LIN {X 0,Y 304.273,Z 903.558,A -85,B 0,C 180,E1 11483.308,E2 11483.308} C_VEL
LIN {X 0,Y 294.742,Z 920.406,A -85,B 0,C 180,E1 11480.364,E2 11480.364} C_VEL
LIN {X 0,Y 285.565,Z 936.169,A -85,B 0,C 180,E1 11477.041,E2 11477.041} C_VEL
LIN {X 0,Y 276.52,Z 951.203,A -85,B 0,C 180,E1 11473.115,E2 11473.115} C_VEL
LIN {X 0,Y 268.033,Z 965.419,A -85,B 0,C 180,E1 11468.539,E2 11468.539} C_VEL
LIN {X 0,Y 261.444,Z 977.018,A -85,B 0,C 180,E1 11463.948,E2 11463.948} C_VEL
LIN {X 0,Y 256.111,Z 986.967,A -85,B 0,C 180,E1 11459.016,E2 11459.016} C_VEL
LIN {X 0,Y 252.21,Z 995.391,A -85,B 0,C 180,E1 11453.857,E2 11453.857} C_VEL
LIN {X 0,Y 249.926,Z 1001.381,A -85,B 0,C 180,E1 11449.156,E2 11449.156} C_VEL
LIN {X 0,Y 248.555,Z 1006.524,A -85,B 0,C 180,E1 11443.973,E2 11443.973} C_VEL
LIN {X 0,Y 248.056,Z 1009.801,A -85,B 0,C 180,E1 11439.05,E2 11439.05} C_VEL
LIN {X 0,Y 247.979,Z 1011.619,A -85,B 0,C 180,E1 11434.631,E2 11434.631} C_VEL
LIN {X 0,Y 248.01,Z 1012.279,A -85,B 0,C 180,E1 11430.006,E2 11430.006} C_VEL
LIN {X 0,Y 247.985,Z 1011.616,A -85,B 0,C 180,E1 11425.613,E2 11425.613} C_VEL
LIN {X 0,Y 248.04,Z 1010.062,A -85,B 0,C 180,E1 11421.662,E2 11421.662} C_VEL
LIN {X 0,Y 248.437,Z 1006.899,A -85,B 0,C 180,E1 11416.745,E2 11416.745} C_VEL
LIN {X 0,Y 249.642,Z 1001.922,A -85,B 0,C 180,E1 11411.661,E2 11411.661} C_VEL
LIN {X 0,Y 251.901,Z 995.507,A -85,B 0,C 180,E1 11406.621,E2 11406.621} C_VEL
LIN {X 0,Y 255.374,Z 987.384,A -85,B 0,C 180,E1 11401.73,E2 11401.73} C_VEL
LIN {X 0,Y 260.313,Z 977.41,A -85,B 0,C 180,E1 11396.858,E2 11396.858} C_VEL
LIN {X 0,Y 266.131,Z 966.36,A -85,B 0,C 180,E1 11392.518,E2 11392.518} C_VEL
LIN {X 0,Y 273.329,Z 953.138,A -85,B 0,C 180,E1 11388.265,E2 11388.265} C_VEL
LIN {X 0,Y 280.892,Z 939.326,A -85,B 0,C 180,E1 11384.619,E2 11384.619} C_VEL
LIN {X 0,Y 289.162,Z 923.71,A -85,B 0,C 180,E1 11381.24,E2 11381.24} C_VEL
LIN {X 0,Y 297.792,Z 906.857,A -85,B 0,C 180,E1 11378.228,E2 11378.228} C_VEL
LIN {X 0,Y 306.271,Z 888.986,A -85,B 0,C 180,E1 11375.632,E2 11375.632} C_VEL
LIN {X 0,Y 315.015,Z 869.115,A -85,B 0,C 180,E1 11373.255,E2 11373.255} C_VEL
LIN {X 0,Y 322.317,Z 850.844,A -85,B 0,C 180,E1 11371.465,E2 11371.465} C_VEL
LIN {X 0,Y 329.921,Z 829.463,A -85,B 0,C 180,E1 11369.755,E2 11369.755} C_VEL
LIN {X 0,Y 336.089,Z 809.722,A -85,B 0,C 180,E1 11368.478,E2 11368.478} C_VEL
LIN {X 0,Y 342.074,Z 787.076,A -85,B 0,C 180,E1 11367.319,E2 11367.319} C_VEL
LIN {X 0,Y 346.854,Z 765.41,A -85,B 0,C 180,E1 11366.46,E2 11366.46} C_VEL
LIN {X 0,Y 350.707,Z 741.944,A -85,B 0,C 180,E1 11365.771,E2 11365.771} C_VEL
LIN {X 0,Y 353.504,Z 715.417,A -85,B 0,C 180,E1 11365.165,E2 11365.165} C_VEL
LIN {X 0,Y 368.316,Z 537.41,A -85,B 0,C 180,E1 11361.544,E2 11361.544} C_VEL
LIN {X 0,Y 362.237,Z 527.156,A -85,B 0,C 180,E1 11359.008,E2 11359.008} C_VEL
LIN {X 0,Y 356.566,Z 518.193,A -85,B 0,C 180,E1 11356.41,E2 11356.41} C_VEL
LIN {X 0,Y 349.782,Z 508.754,A -85,B 0,C 180,E1 11352.967,E2 11352.967} C_VEL
LIN {X 0,Y 345.656,Z 503.263,A -85,B 0,C 180,E1 11350.584,E2 11350.584} C_VEL
LIN {X 0,Y 341.9,Z 498.285,A -85,B 0,C 180,E1 11348.153,E2 11348.153} C_VEL
LIN {X 0,Y 338.19,Z 493.354,A -85,B 0,C 180,E1 11345.428,E2 11345.428} C_VEL
LIN {X 0,Y 334.542,Z 488.626,A -85,B 0,C 180,E1 11342.312,E2 11342.312} C_VEL
LIN {X 0,Y 330.628,Z 484.034,A -85,B 0,C 180,E1 11338.18,E2 11338.18} C_VEL
LIN {X 0,Y 329.692,Z 482.187,A -85,B 0,C 180,E1 11336.87,E2 11336.87} C_VEL
LIN {X 0,Y 326.46,Z 479.325,A -85,B 0,C 180,E1 11331.546,E2 11331.546} C_VEL
LIN {X 0,Y 325.3,Z 476.564,A -85,B 0,C 180,E1 11327.394,E2 11327.394} C_VEL
LIN {X 0,Y 324.939,Z 476.13,A -85,B 0,C 180,E1 11322.449,E2 11322.449} C_VEL
LIN {X 0,Y 325.484,Z 476.933,A -85,B 0,C 180,E1 11318.935,E2 11318.935} C_VEL
LIN {X 0,Y 327.95,Z 481.052,A -85,B 0,C 180,E1 11312.785,E2 11312.785} C_VEL
LIN {X 0,Y 329.949,Z 482.531,A -85,B 0,C 180,E1 11309.999,E2 11309.999} C_VEL
LIN {X 0,Y 332.367,Z 486.461,A -85,B 0,C 180,E1 11307.009,E2 11307.009} C_VEL
LIN {X 0,Y 334.594,Z 488.635,A -85,B 0,C 180,E1 11304.883,E2 11304.883} C_VEL
LIN {X 0,Y 338.152,Z 493.293,A -85,B 0,C 180,E1 11301.831,E2 11301.831} C_VEL
LIN {X 0,Y 343.422,Z 500.232,A -85,B 0,C 180,E1 11298.073,E2 11298.073} C_VEL
LIN {X 0,Y 347.643,Z 505.888,A -85,B 0,C 180,E1 11295.494,E2 11295.494} C_VEL
LIN {X 0,Y 351.997,Z 511.892,A -85,B 0,C 180,E1 11293.112,E2 11293.112} C_VEL
LIN {X 0,Y 358.041,Z 520.377,A -85,B 0,C 180,E1 11290.165,E2 11290.165} C_VEL
LIN {X 0,Y 364.276,Z 529.62,A -85,B 0,C 180,E1 11287.445,E2 11287.445} C_VEL
LIN {X 0,Y 367.903,Z 535.336,A -85,B 0,C 180,E1 11285.985,E2 11285.985} C_VEL
LIN {X 0,Y 352.417,Z 718.617,A -85,B 0,C 180,E1 11282.246,E2 11282.246} C_VEL
LIN {X 0,Y 348.99,Z 742.464,A -85,B 0,C 180,E1 11281.584,E2 11281.584} C_VEL
LIN {X 0,Y 344.711,Z 764.957,A -85,B 0,C 180,E1 11280.739,E2 11280.739} C_VEL
LIN {X 0,Y 339.382,Z 786.794,A -85,B 0,C 180,E1 11279.66,E2 11279.66} C_VEL
LIN {X 0,Y 333.081,Z 808.628,A -85,B 0,C 180,E1 11278.307,E2 11278.307} C_VEL
LIN {X 0,Y 326.617,Z 827.813,A -85,B 0,C 180,E1 11276.836,E2 11276.836} C_VEL
LIN {X 0,Y 318.314,Z 849.468,A -85,B 0,C 180,E1 11274.798,E2 11274.798} C_VEL
LIN {X 0,Y 310.335,Z 868.235,A -85,B 0,C 180,E1 11272.638,E2 11272.638} C_VEL
LIN {X 0,Y 301.952,Z 886,A -85,B 0,C 180,E1 11270.138,E2 11270.138} C_VEL
LIN {X 0,Y 293.398,Z 903.061,A -85,B 0,C 180,E1 11267.241,E2 11267.241} C_VEL
LIN {X 0,Y 285.468,Z 917.802,A -85,B 0,C 180,E1 11264.186,E2 11264.186} C_VEL
LIN {X 0,Y 277.047,Z 932.922,A -85,B 0,C 180,E1 11260.39,E2 11260.39} C_VEL
LIN {X 0,Y 270.038,Z 945.31,A -85,B 0,C 180,E1 11256.585,E2 11256.585} C_VEL
LIN {X 0,Y 263.418,Z 957.018,A -85,B 0,C 180,E1 11252.17,E2 11252.17} C_VEL
LIN {X 0,Y 258.058,Z 966.993,A -85,B 0,C 180,E1 11247.552,E2 11247.552} C_VEL
LIN {X 0,Y 253.931,Z 975.148,A -85,B 0,C 180,E1 11242.756,E2 11242.756} C_VEL
LIN {X 0,Y 251.035,Z 981.913,A -85,B 0,C 180,E1 11237.808,E2 11237.808} C_VEL
LIN {X 0,Y 249.276,Z 986.831,A -85,B 0,C 180,E1 11232.968,E2 11232.968} C_VEL
LIN {X 0,Y 248.412,Z 990.387,A -85,B 0,C 180,E1 11228.26,E2 11228.26} C_VEL
LIN {X 0,Y 248.06,Z 992.643,A -85,B 0,C 180,E1 11223.417,E2 11223.417} C_VEL
LIN {X 0,Y 248.003,Z 993.532,A -85,B 0,C 180,E1 11219.464,E2 11219.464} C_VEL
LIN {X 0,Y 248.018,Z 993.558,A -85,B 0,C 180,E1 11215.327,E2 11215.327} C_VEL
LIN {X 0,Y 248.208,Z 992.348,A -85,B 0,C 180,E1 11210.302,E2 11210.302} C_VEL
LIN {X 0,Y 248.763,Z 989.901,A -85,B 0,C 180,E1 11205.618,E2 11205.618} C_VEL
LIN {X 0,Y 250.147,Z 986.027,A -85,B 0,C 180,E1 11200.578,E2 11200.578} C_VEL
LIN {X 0,Y 252.048,Z 981.677,A -85,B 0,C 180,E1 11196.478,E2 11196.478} C_VEL
LIN {X 0,Y 252.075,Z 979.727,A -85,B 0,C 180,E1 11194.77,E2 11194.77} C_VEL
LIN {X 0,Y 249.469,Z 974.34,A -85,B 0,C 180,E1 11189.975,E2 11189.975} C_VEL
LIN {X 0,Y 250.083,Z 972.352,A -85,B 0,C 180,E1 11188.654,E2 11188.654} C_VEL
LIN {X 0,Y 255.769,Z 963.603,A -85,B 0,C 180,E1 11183.819,E2 11183.819} C_VEL
LIN {X 0,Y 263.044,Z 952.8,A -85,B 0,C 180,E1 11179.081,E2 11179.081} C_VEL
LIN {X 0,Y 271.121,Z 941.127,A -85,B 0,C 180,E1 11174.921,E2 11174.921} C_VEL
LIN {X 0,Y 280.187,Z 927.63,A -85,B 0,C 180,E1 11171.066,E2 11171.066} C_VEL
LIN {X 0,Y 290.421,Z 912.011,A -85,B 0,C 180,E1 11167.442,E2 11167.442} C_VEL
LIN {X 0,Y 300.488,Z 895.774,A -85,B 0,C 180,E1 11164.39,E2 11164.39} C_VEL
LIN {X 0,Y 310.818,Z 877.793,A -85,B 0,C 180,E1 11161.66,E2 11161.66} C_VEL
LIN {X 0,Y 320.673,Z 859.276,A -85,B 0,C 180,E1 11159.366,E2 11159.366} C_VEL
LIN {X 0,Y 329.619,Z 840.558,A -85,B 0,C 180,E1 11157.48,E2 11157.48} C_VEL
LIN {X 0,Y 338.92,Z 818.761,A -85,B 0,C 180,E1 11155.701,E2 11155.701} C_VEL
LIN {X 0,Y 346.656,Z 797.924,A -85,B 0,C 180,E1 11154.339,E2 11154.339} C_VEL
LIN {X 0,Y 353.44,Z 776.189,A -85,B 0,C 180,E1 11153.215,E2 11153.215} C_VEL
LIN {X 0,Y 359.373,Z 753.167,A -85,B 0,C 180,E1 11152.29,E2 11152.29} C_VEL
LIN {X 0,Y 363.773,Z 730.744,A -85,B 0,C 180,E1 11151.624,E2 11151.624} C_VEL
LIN {X 0,Y 367.924,Z 699.697,A -85,B 0,C 180,E1 11150.938,E2 11150.938} C_VEL
LIN {X 0,Y 385.975,Z 550.691,A -85,B 0,C 180,E1 11147.888,E2 11147.888} C_VEL
LIN {X 0,Y 385.47,Z 549.203,A -85,B 0,C 180,E1 11146.806,E2 11146.806} C_VEL
LIN {X 0,Y 385.143,Z 546.456,A -85,B 0,C 180,E1 11144.182,E2 11144.182} C_VEL
LIN {X 0,Y 385.911,Z 550.412,A -85,B 0,C 180,E1 11140.711,E2 11140.711} C_VEL
LIN {X 0,Y 385.992,Z 551.133,A -85,B 0,C 180,E1 11140.47,E2 11140.47} C_VEL
LIN {X 0,Y 364.137,Z 730.975,A -85,B 0,C 180,E1 11136.773,E2 11136.773} C_VEL
LIN {X 0,Y 359.583,Z 754.878,A -85,B 0,C 180,E1 11136.149,E2 11136.149} C_VEL
LIN {X 0,Y 353.483,Z 779.088,A -85,B 0,C 180,E1 11135.33,E2 11135.33} C_VEL
LIN {X 0,Y 347.082,Z 800.029,A -85,B 0,C 180,E1 11134.385,E2 11134.385} C_VEL
LIN {X 0,Y 338.752,Z 822.956,A -85,B 0,C 180,E1 11133.053,E2 11133.053} C_VEL
LIN {X 0,Y 330.353,Z 843.418,A -85,B 0,C 180,E1 11131.556,E2 11131.556} C_VEL
LIN {X 0,Y 320.737,Z 863.996,A -85,B 0,C 180,E1 11129.668,E2 11129.668} C_VEL
LIN {X 0,Y 310.127,Z 884.727,A -85,B 0,C 180,E1 11127.302,E2 11127.302} C_VEL
LIN {X 0,Y 300.566,Z 902.017,A -85,B 0,C 180,E1 11124.866,E2 11124.866} C_VEL
LIN {X 0,Y 290.679,Z 918.803,A -85,B 0,C 180,E1 11121.977,E2 11121.977} C_VEL
LIN {X 0,Y 281.002,Z 934.642,A -85,B 0,C 180,E1 11118.663,E2 11118.663} C_VEL
LIN {X 0,Y 271.827,Z 949.086,A -85,B 0,C 180,E1 11114.935,E2 11114.935} C_VEL
LIN {X 0,Y 263.456,Z 962.405,A -85,B 0,C 180,E1 11110.756,E2 11110.756} C_VEL
LIN {X 0,Y 256.07,Z 974.241,A -85,B 0,C 180,E1 11106.134,E2 11106.134} C_VEL
LIN {X 0,Y 249.713,Z 985.187,A -85,B 0,C 180,E1 11100.837,E2 11100.837} C_VEL
LIN {X 0,Y 245.409,Z 993.524,A -85,B 0,C 180,E1 11095.79,E2 11095.79} C_VEL
LIN {X 0,Y 242.345,Z 1000.596,A -85,B 0,C 180,E1 11090.283,E2 11090.283} C_VEL
LIN {X 0,Y 240.814,Z 1005.415,A -85,B 0,C 180,E1 11085.416,E2 11085.416} C_VEL
LIN {X 0,Y 240.093,Z 1009.147,A -85,B 0,C 180,E1 11080.079,E2 11080.079} C_VEL
LIN {X 0,Y 239.984,Z 1011.027,A -85,B 0,C 180,E1 11075.745,E2 11075.745} C_VEL
LIN {X 0,Y 240.009,Z 1011.89,A -85,B 0,C 180,E1 11071.438,E2 11071.438} C_VEL
LIN {X 0,Y 239.983,Z 1011.699,A -85,B 0,C 180,E1 11066.902,E2 11066.902} C_VEL
LIN {X 0,Y 240.012,Z 1010.078,A -85,B 0,C 180,E1 11062.105,E2 11062.105} C_VEL
LIN {X 0,Y 240.29,Z 1007.547,A -85,B 0,C 180,E1 11057.755,E2 11057.755} C_VEL
LIN {X 0,Y 241.318,Z 1003.277,A -85,B 0,C 180,E1 11052.65,E2 11052.65} C_VEL
LIN {X 0,Y 243.351,Z 997.323,A -85,B 0,C 180,E1 11047.543,E2 11047.543} C_VEL
LIN {X 0,Y 246.829,Z 989.456,A -85,B 0,C 180,E1 11042.243,E2 11042.243} C_VEL
LIN {X 0,Y 251.362,Z 980.468,A -85,B 0,C 180,E1 11037.487,E2 11037.487} C_VEL
LIN {X 0,Y 257.793,Z 968.775,A -85,B 0,C 180,E1 11032.497,E2 11032.497} C_VEL
LIN {X 0,Y 264.669,Z 956.756,A -85,B 0,C 180,E1 11028.336,E2 11028.336} C_VEL
LIN {X 0,Y 272.719,Z 942.628,A -85,B 0,C 180,E1 11024.373,E2 11024.373} C_VEL
LIN {X 0,Y 281.372,Z 927.213,A -85,B 0,C 180,E1 11020.819,E2 11020.819} C_VEL
LIN {X 0,Y 290.123,Z 910.743,A -85,B 0,C 180,E1 11017.738,E2 11017.738} C_VEL
LIN {X 0,Y 299.647,Z 891.763,A -85,B 0,C 180,E1 11014.842,E2 11014.842} C_VEL
LIN {X 0,Y 307.897,Z 873.95,A -85,B 0,C 180,E1 11012.619,E2 11012.619} C_VEL
LIN {X 0,Y 316.167,Z 854.185,A -85,B 0,C 180,E1 11010.607,E2 11010.607} C_VEL
LIN {X 0,Y 323.936,Z 833.646,A -85,B 0,C 180,E1 11008.894,E2 11008.894} C_VEL
LIN {X 0,Y 330.427,Z 813.727,A -85,B 0,C 180,E1 11007.564,E2 11007.564} C_VEL
LIN {X 0,Y 336.539,Z 792.368,A -85,B 0,C 180,E1 11006.408,E2 11006.408} C_VEL
LIN {X 0,Y 341.563,Z 770.746,A -85,B 0,C 180,E1 11005.509,E2 11005.509} C_VEL
LIN {X 0,Y 345.978,Z 746.91,A -85,B 0,C 180,E1 11004.761,E2 11004.761} C_VEL
LIN {X 0,Y 348.781,Z 724.177,A -85,B 0,C 180,E1 11004.211,E2 11004.211} C_VEL
LIN {X 0,Y 364.397,Z 541.876,A -85,B 0,C 180,E1 11000.498,E2 11000.498} C_VEL
LIN {X 0,Y 357.482,Z 530.256,A -85,B 0,C 180,E1 10997.455,E2 10997.455} C_VEL
LIN {X 0,Y 353.106,Z 523.64,A -85,B 0,C 180,E1 10995.352,E2 10995.352} C_VEL
LIN {X 0,Y 347.215,Z 515.344,A -85,B 0,C 180,E1 10992.219,E2 10992.219} C_VEL
LIN {X 0,Y 343.719,Z 510.585,A -85,B 0,C 180,E1 10990.136,E2 10990.136} C_VEL
LIN {X 0,Y 340.272,Z 505.911,A -85,B 0,C 180,E1 10987.853,E2 10987.853} C_VEL
LIN {X 0,Y 336.497,Z 500.899,A -85,B 0,C 180,E1 10985.028,E2 10985.028} C_VEL
LIN {X 0,Y 332.589,Z 495.69,A -85,B 0,C 180,E1 10981.55,E2 10981.55} C_VEL
LIN {X 0,Y 329.472,Z 492.131,A -85,B 0,C 180,E1 10978.173,E2 10978.173} C_VEL
LIN {X 0,Y 328.272,Z 489.964,A -85,B 0,C 180,E1 10976.507,E2 10976.507} C_VEL
LIN {X 0,Y 325.025,Z 486.819,A -85,B 0,C 180,E1 10970.795,E2 10970.795} C_VEL
LIN {X 0,Y 324.17,Z 484.48,A -85,B 0,C 180,E1 10967.35,E2 10967.35} C_VEL
LIN {X 0,Y 323.822,Z 484.058,A -85,B 0,C 180,E1 10962.386,E2 10962.386} C_VEL
LIN {X 0,Y 324.331,Z 484.829,A -85,B 0,C 180,E1 10959.046,E2 10959.046} C_VEL
LIN {X 0,Y 326.772,Z 488.949,A -85,B 0,C 180,E1 10952.876,E2 10952.876} C_VEL
LIN {X 0,Y 328.682,Z 490.428,A -85,B 0,C 180,E1 10950.173,E2 10950.173} C_VEL
LIN {X 0,Y 331.187,Z 494.423,A -85,B 0,C 180,E1 10947.053,E2 10947.053} C_VEL
LIN {X 0,Y 333.166,Z 496.407,A -85,B 0,C 180,E1 10945.13,E2 10945.13} C_VEL
LIN {X 0,Y 336.817,Z 501.145,A -85,B 0,C 180,E1 10941.977,E2 10941.977} C_VEL
LIN {X 0,Y 341.825,Z 507.961,A -85,B 0,C 180,E1 10938.338,E2 10938.338} C_VEL
LIN {X 0,Y 345.942,Z 513.558,A -85,B 0,C 180,E1 10935.781,E2 10935.781} C_VEL
LIN {X 0,Y 351.701,Z 521.468,A -85,B 0,C 180,E1 10932.641,E2 10932.641} C_VEL
LIN {X 0,Y 359.446,Z 532.869,A -85,B 0,C 180,E1 10928.969,E2 10928.969} C_VEL
LIN {X 0,Y 363.986,Z 540.116,A -85,B 0,C 180,E1 10927.02,E2 10927.02} C_VEL
LIN {X 0,Y 348.486,Z 718.572,A -85,B 0,C 180,E1 10923.389,E2 10923.389} C_VEL
LIN {X 0,Y 344.983,Z 742.486,A -85,B 0,C 180,E1 10922.732,E2 10922.732} C_VEL
LIN {X 0,Y 340.764,Z 764.299,A -85,B 0,C 180,E1 10921.924,E2 10921.924} C_VEL
LIN {X 0,Y 335.288,Z 786.305,A -85,B 0,C 180,E1 10920.852,E2 10920.852} C_VEL
LIN {X 0,Y 328.812,Z 808.306,A -85,B 0,C 180,E1 10919.506,E2 10919.506} C_VEL
LIN {X 0,Y 321.846,Z 828.447,A -85,B 0,C 180,E1 10917.97,E2 10917.97} C_VEL
LIN {X 0,Y 313.573,Z 849.47,A -85,B 0,C 180,E1 10915.998,E2 10915.998} C_VEL
LIN {X 0,Y 305.368,Z 868.244,A -85,B 0,C 180,E1 10913.846,E2 10913.846} C_VEL
LIN {X 0,Y 296.691,Z 886.068,A -85,B 0,C 180,E1 10911.338,E2 10911.338} C_VEL
LIN {X 0,Y 287.806,Z 903.177,A -85,B 0,C 180,E1 10908.423,E2 10908.423} C_VEL
LIN {X 0,Y 279.56,Z 917.965,A -85,B 0,C 180,E1 10905.341,E2 10905.341} C_VEL
LIN {X 0,Y 270.774,Z 933.145,A -85,B 0,C 180,E1 10901.496,E2 10901.496} C_VEL
LIN {X 0,Y 263.418,Z 945.55,A -85,B 0,C 180,E1 10897.628,E2 10897.628} C_VEL
LIN {X 0,Y 256.448,Z 957.27,A -85,B 0,C 180,E1 10893.123,E2 10893.123} C_VEL
LIN {X 0,Y 250.781,Z 967.271,A -85,B 0,C 180,E1 10888.395,E2 10888.395} C_VEL
LIN {X 0,Y 246.391,Z 975.442,A -85,B 0,C 180,E1 10883.47,E2 10883.47} C_VEL
LIN {X 0,Y 243.29,Z 982.204,A -85,B 0,C 180,E1 10878.377,E2 10878.377} C_VEL
LIN {X 0,Y 241.397,Z 987.121,A -85,B 0,C 180,E1 10873.388,E2 10873.388} C_VEL
LIN {X 0,Y 240.452,Z 990.68,A -85,B 0,C 180,E1 10868.53,E2 10868.53} C_VEL
LIN {X 0,Y 240.069,Z 992.939,A -85,B 0,C 180,E1 10863.53,E2 10863.53} C_VEL
LIN {X 0,Y 240.009,Z 993.831,A -85,B 0,C 180,E1 10859.447,E2 10859.447} C_VEL
LIN {X 0,Y 240.028,Z 993.865,A -85,B 0,C 180,E1 10855.196,E2 10855.196} C_VEL
LIN {X 0,Y 240.246,Z 992.659,A -85,B 0,C 180,E1 10849.977,E2 10849.977} C_VEL
LIN {X 0,Y 240.869,Z 990.205,A -85,B 0,C 180,E1 10845.109,E2 10845.109} C_VEL
LIN {X 0,Y 242.472,Z 986.181,A -85,B 0,C 180,E1 10839.73,E2 10839.73} C_VEL
LIN {X 0,Y 245.299,Z 980.443,A -85,B 0,C 180,E1 10834.393,E2 10834.393} C_VEL
LIN {X 0,Y 249.769,Z 972.881,A -85,B 0,C 180,E1 10828.973,E2 10828.973} C_VEL
LIN {X 0,Y 250.083,Z 972.352,A -85,B 0,C 180,E1 10828.654,E2 10828.654} C_VEL
LIN {X 0,Y 250.83,Z 969.842,A -85,B 0,C 180,E1 10826.984,E2 10826.984} C_VEL
LIN {X 0,Y 250.309,Z 963.175,A -85,B 0,C 180,E1 10822.369,E2 10822.369} C_VEL
LIN {X 0,Y 251.566,Z 960.534,A -85,B 0,C 180,E1 10821,E2 10821} C_VEL
LIN {X 0,Y 259.746,Z 949.363,A -85,B 0,C 180,E1 10816.321,E2 10816.321} C_VEL
LIN {X 0,Y 268.558,Z 937.101,A -85,B 0,C 180,E1 10812.253,E2 10812.253} C_VEL
LIN {X 0,Y 278.488,Z 923.122,A -85,B 0,C 180,E1 10808.466,E2 10808.466} C_VEL
LIN {X 0,Y 288.681,Z 907.98,A -85,B 0,C 180,E1 10805.167,E2 10805.167} C_VEL
LIN {X 0,Y 299.739,Z 890.56,A -85,B 0,C 180,E1 10802.103,E2 10802.103} C_VEL
LIN {X 0,Y 310.391,Z 872.535,A -85,B 0,C 180,E1 10799.539,E2 10799.539} C_VEL
LIN {X 0,Y 320.299,Z 853.861,A -85,B 0,C 180,E1 10797.402,E2 10797.402} C_VEL
LIN {X 0,Y 329.782,Z 834.246,A -85,B 0,C 180,E1 10795.566,E2 10795.566} C_VEL
LIN {X 0,Y 337.983,Z 814.98,A -85,B 0,C 180,E1 10794.105,E2 10794.105} C_VEL
LIN {X 0,Y 346.025,Z 793.278,A -85,B 0,C 180,E1 10792.78,E2 10792.78} C_VEL
LIN {X 0,Y 352.086,Z 774.015,A -85,B 0,C 180,E1 10791.837,E2 10791.837} C_VEL
LIN {X 0,Y 358.241,Z 749.963,A -85,B 0,C 180,E1 10790.927,E2 10790.927} C_VEL
LIN {X 0,Y 362.722,Z 727.263,A -85,B 0,C 180,E1 10790.295,E2 10790.295} C_VEL
LIN {X 0,Y 368.453,Z 682.596,A -85,B 0,C 180,E1 10789.357,E2 10789.357} C_VEL
LIN {X 0,Y 384.347,Z 557.233,A -85,B 0,C 180,E1 10786.843,E2 10786.843} C_VEL
LIN {X 0,Y 384.004,Z 554.448,A -85,B 0,C 180,E1 10784.134,E2 10784.134} C_VEL
LIN {X 0,Y 384.355,Z 557.383,A -85,B 0,C 180,E1 10781.538,E2 10781.538} C_VEL
LIN {X 0,Y 362.49,Z 730.382,A -85,B 0,C 180,E1 10778.025,E2 10778.025} C_VEL
LIN {X 0,Y 357.809,Z 754.212,A -85,B 0,C 180,E1 10777.417,E2 10777.417} C_VEL
LIN {X 0,Y 351.572,Z 778.344,A -85,B 0,C 180,E1 10776.625,E2 10776.625} C_VEL
LIN {X 0,Y 345.398,Z 797.974,A -85,B 0,C 180,E1 10775.77,E2 10775.77} C_VEL
LIN {X 0,Y 336.833,Z 821.09,A -85,B 0,C 180,E1 10774.481,E2 10774.481} C_VEL
LIN {X 0,Y 328.902,Z 839.849,A -85,B 0,C 180,E1 10773.162,E2 10773.162} C_VEL
LIN {X 0,Y 319.027,Z 860.66,A -85,B 0,C 180,E1 10771.347,E2 10771.347} C_VEL
LIN {X 0,Y 308.867,Z 880.159,A -85,B 0,C 180,E1 10769.239,E2 10769.239} C_VEL
LIN {X 0,Y 297.98,Z 899.113,A -85,B 0,C 180,E1 10766.675,E2 10766.675} C_VEL
LIN {X 0,Y 287.111,Z 916.922,A -85,B 0,C 180,E1 10763.7,E2 10763.7} C_VEL
LIN {X 0,Y 277.217,Z 932.312,A -85,B 0,C 180,E1 10760.526,E2 10760.526} C_VEL
LIN {X 0,Y 266.963,Z 947.738,A -85,B 0,C 180,E1 10756.607,E2 10756.607} C_VEL
LIN {X 0,Y 258.001,Z 961.15,A -85,B 0,C 180,E1 10752.407,E2 10752.407} C_VEL
LIN {X 0,Y 250.031,Z 973.089,A -85,B 0,C 180,E1 10747.729,E2 10747.729} C_VEL
LIN {X 0,Y 243.358,Z 983.761,A -85,B 0,C 180,E1 10742.569,E2 10742.569} C_VEL
LIN {X 0,Y 238.548,Z 992.131,A -85,B 0,C 180,E1 10737.461,E2 10737.461} C_VEL
LIN {X 0,Y 234.849,Z 999.822,A -85,B 0,C 180,E1 10731.484,E2 10731.484} C_VEL
LIN {X 0,Y 233.046,Z 1004.722,A -85,B 0,C 180,E1 10726.455,E2 10726.455} C_VEL
LIN {X 0,Y 232.151,Z 1008.636,A -85,B 0,C 180,E1 10720.899,E2 10720.899} C_VEL
LIN {X 0,Y 231.995,Z 1010.665,A -85,B 0,C 180,E1 10716.192,E2 10716.192} C_VEL
LIN {X 0,Y 232.013,Z 1011.539,A -85,B 0,C 180,E1 10711.982,E2 10711.982} C_VEL
LIN {X 0,Y 232.004,Z 1011.463,A -85,B 0,C 180,E1 10707.537,E2 10707.537} C_VEL
LIN {X 0,Y 231.992,Z 1010.091,A -85,B 0,C 180,E1 10702.578,E2 10702.578} C_VEL
LIN {X 0,Y 232.279,Z 1007.526,A -85,B 0,C 180,E1 10697.831,E2 10697.831} C_VEL
LIN {X 0,Y 233.252,Z 1003.589,A -85,B 0,C 180,E1 10692.803,E2 10692.803} C_VEL
LIN {X 0,Y 235.433,Z 997.533,A -85,B 0,C 180,E1 10687.273,E2 10687.273} C_VEL
LIN {X 0,Y 238.878,Z 990.165,A -85,B 0,C 180,E1 10682.026,E2 10682.026} C_VEL
LIN {X 0,Y 243.732,Z 980.987,A -85,B 0,C 180,E1 10676.943,E2 10676.943} C_VEL
LIN {X 0,Y 249.785,Z 970.586,A -85,B 0,C 180,E1 10672.243,E2 10672.243} C_VEL
LIN {X 0,Y 256.792,Z 958.763,A -85,B 0,C 180,E1 10667.965,E2 10667.965} C_VEL
LIN {X 0,Y 265.004,Z 945.103,A -85,B 0,C 180,E1 10663.903,E2 10663.903} C_VEL
LIN {X 0,Y 273.321,Z 930.893,A -85,B 0,C 180,E1 10660.467,E2 10660.467} C_VEL
LIN {X 0,Y 283.046,Z 913.515,A -85,B 0,C 180,E1 10657.039,E2 10657.039} C_VEL
LIN {X 0,Y 292.16,Z 896.275,A -85,B 0,C 180,E1 10654.273,E2 10654.273} C_VEL
LIN {X 0,Y 301.237,Z 877.478,A -85,B 0,C 180,E1 10651.833,E2 10651.833} C_VEL
LIN {X 0,Y 310.163,Z 857.326,A -85,B 0,C 180,E1 10649.697,E2 10649.697} C_VEL
LIN {X 0,Y 317.85,Z 837.796,A -85,B 0,C 180,E1 10648.023,E2 10648.023} C_VEL
LIN {X 0,Y 325.61,Z 815.251,A -85,B 0,C 180,E1 10646.472,E2 10646.472} C_VEL
LIN {X 0,Y 331.814,Z 794.283,A -85,B 0,C 180,E1 10645.327,E2 10645.327} C_VEL
LIN {X 0,Y 337.241,Z 771.894,A -85,B 0,C 180,E1 10644.384,E2 10644.384} C_VEL
LIN {X 0,Y 341.774,Z 748.578,A -85,B 0,C 180,E1 10643.643,E2 10643.643} C_VEL
LIN {X 0,Y 344.775,Z 725.283,A -85,B 0,C 180,E1 10643.077,E2 10643.077} C_VEL
LIN {X 0,Y 360.639,Z 546.513,A -85,B 0,C 180,E1 10639.451,E2 10639.451} C_VEL
LIN {X 0,Y 353.388,Z 534.361,A -85,B 0,C 180,E1 10636.097,E2 10636.097} C_VEL
LIN {X 0,Y 347.855,Z 526.352,A -85,B 0,C 180,E1 10633.251,E2 10633.251} C_VEL
LIN {X 0,Y 342.46,Z 518.686,A -85,B 0,C 180,E1 10630.088,E2 10630.088} C_VEL
LIN {X 0,Y 338.412,Z 513.267,A -85,B 0,C 180,E1 10627.384,E2 10627.384} C_VEL
LIN {X 0,Y 334.93,Z 508.541,A -85,B 0,C 180,E1 10624.708,E2 10624.708} C_VEL
LIN {X 0,Y 331.095,Z 503.387,A -85,B 0,C 180,E1 10621.211,E2 10621.211} C_VEL
LIN {X 0,Y 328.068,Z 499.745,A -85,B 0,C 180,E1 10617.816,E2 10617.816} C_VEL
LIN {X 0,Y 326.997,Z 497.816,A -85,B 0,C 180,E1 10616.318,E2 10616.318} C_VEL
LIN {X 0,Y 323.761,Z 494.524,A -85,B 0,C 180,E1 10610.4,E2 10610.4} C_VEL
LIN {X 0,Y 323.009,Z 492.363,A -85,B 0,C 180,E1 10607.122,E2 10607.122} C_VEL
LIN {X 0,Y 322.706,Z 491.987,A -85,B 0,C 180,E1 10602.323,E2 10602.323} C_VEL
LIN {X 0,Y 323.191,Z 492.765,A -85,B 0,C 180,E1 10599.097,E2 10599.097} C_VEL
LIN {X 0,Y 325.622,Z 496.873,A -85,B 0,C 180,E1 10592.919,E2 10592.919} C_VEL
LIN {X 0,Y 327.409,Z 498.32,A -85,B 0,C 180,E1 10590.348,E2 10590.348} C_VEL
LIN {X 0,Y 330.068,Z 502.444,A -85,B 0,C 180,E1 10587.034,E2 10587.034} C_VEL
LIN {X 0,Y 331.775,Z 504.232,A -85,B 0,C 180,E1 10585.348,E2 10585.348} C_VEL
LIN {X 0,Y 336.151,Z 510.108,A -85,B 0,C 180,E1 10581.562,E2 10581.562} C_VEL
LIN {X 0,Y 340.168,Z 515.581,A -85,B 0,C 180,E1 10578.653,E2 10578.653} C_VEL
LIN {X 0,Y 344.158,Z 521.086,A -85,B 0,C 180,E1 10576.128,E2 10576.128} C_VEL
LIN {X 0,Y 349.74,Z 528.914,A -85,B 0,C 180,E1 10573.016,E2 10573.016} C_VEL
LIN {X 0,Y 357.171,Z 540.032,A -85,B 0,C 180,E1 10569.409,E2 10569.409} C_VEL
LIN {X 0,Y 360.172,Z 545.076,A -85,B 0,C 180,E1 10568.073,E2 10568.073} C_VEL
LIN {X 0,Y 344.583,Z 719.058,A -85,B 0,C 180,E1 10564.541,E2 10564.541} C_VEL
LIN {X 0,Y 340.993,Z 742.926,A -85,B 0,C 180,E1 10563.888,E2 10563.888} C_VEL
LIN {X 0,Y 336.607,Z 765.023,A -85,B 0,C 180,E1 10563.073,E2 10563.073} C_VEL
LIN {X 0,Y 330.998,Z 786.985,A -85,B 0,C 180,E1 10562.008,E2 10562.008} C_VEL
LIN {X 0,Y 324.26,Z 809.231,A -85,B 0,C 180,E1 10560.649,E2 10560.649} C_VEL
LIN {X 0,Y 317.522,Z 828.202,A -85,B 0,C 180,E1 10559.208,E2 10559.208} C_VEL
LIN {X 0,Y 309.005,Z 849.325,A -85,B 0,C 180,E1 10557.242,E2 10557.242} C_VEL
LIN {X 0,Y 300.826,Z 867.508,A -85,B 0,C 180,E1 10555.172,E2 10555.172} C_VEL
LIN {X 0,Y 291.842,Z 885.55,A -85,B 0,C 180,E1 10552.664,E2 10552.664} C_VEL
LIN {X 0,Y 282.87,Z 902.376,A -85,B 0,C 180,E1 10549.83,E2 10549.83} C_VEL
LIN {X 0,Y 273.766,Z 918.107,A -85,B 0,C 180,E1 10546.545,E2 10546.545} C_VEL
LIN {X 0,Y 265.04,Z 932.627,A -85,B 0,C 180,E1 10542.854,E2 10542.854} C_VEL
LIN {X 0,Y 257.642,Z 944.516,A -85,B 0,C 180,E1 10539.149,E2 10539.149} C_VEL
LIN {X 0,Y 249.874,Z 957.014,A -85,B 0,C 180,E1 10534.354,E2 10534.354} C_VEL
LIN {X 0,Y 243.972,Z 966.785,A -85,B 0,C 180,E1 10529.673,E2 10529.673} C_VEL
LIN {X 0,Y 239.077,Z 975.354,A -85,B 0,C 180,E1 10524.474,E2 10524.474} C_VEL
LIN {X 0,Y 235.692,Z 982.205,A -85,B 0,C 180,E1 10519.236,E2 10519.236} C_VEL
LIN {X 0,Y 233.53,Z 987.411,A -85,B 0,C 180,E1 10513.835,E2 10513.835} C_VEL
LIN {X 0,Y 232.462,Z 991.145,A -85,B 0,C 180,E1 10508.549,E2 10508.549} C_VEL
LIN {X 0,Y 232.07,Z 993.314,A -85,B 0,C 180,E1 10503.373,E2 10503.373} C_VEL
LIN {X 0,Y 232.023,Z 994.163,A -85,B 0,C 180,E1 10499.143,E2 10499.143} C_VEL
LIN {X 0,Y 232.05,Z 994.137,A -85,B 0,C 180,E1 10494.526,E2 10494.526} C_VEL
LIN {X 0,Y 232.308,Z 992.768,A -85,B 0,C 180,E1 10489.133,E2 10489.133} C_VEL
LIN {X 0,Y 233.072,Z 990.318,A -85,B 0,C 180,E1 10484.233,E2 10484.233} C_VEL
LIN {X 0,Y 235.044,Z 985.909,A -85,B 0,C 180,E1 10478.395,E2 10478.395} C_VEL
LIN {X 0,Y 238.032,Z 980.515,A -85,B 0,C 180,E1 10473.282,E2 10473.282} C_VEL
LIN {X 0,Y 243.262,Z 972.364,A -85,B 0,C 180,E1 10467.392,E2 10467.392} C_VEL
LIN {X 0,Y 249.653,Z 963.285,A -85,B 0,C 180,E1 10462.298,E2 10462.298} C_VEL
LIN {X 0,Y 251.566,Z 960.534,A -85,B 0,C 180,E1 10461,E2 10461} C_VEL
LIN {X 0,Y 253.069,Z 957.47,A -85,B 0,C 180,E1 10459.419,E2 10459.419} C_VEL
LIN {X 0,Y 254.676,Z 949.444,A -85,B 0,C 180,E1 10454.996,E2 10454.996} C_VEL
LIN {X 0,Y 256.52,Z 946.309,A -85,B 0,C 180,E1 10453.74,E2 10453.74} C_VEL
LIN {X 0,Y 266.136,Z 933.778,A -85,B 0,C 180,E1 10449.734,E2 10449.734} C_VEL
LIN {X 0,Y 276.545,Z 919.522,A -85,B 0,C 180,E1 10446.104,E2 10446.104} C_VEL
LIN {X 0,Y 287.823,Z 903.397,A -85,B 0,C 180,E1 10442.788,E2 10442.788} C_VEL
LIN {X 0,Y 298.38,Z 887.154,A -85,B 0,C 180,E1 10440.097,E2 10440.097} C_VEL
LIN {X 0,Y 309.548,Z 868.48,A -85,B 0,C 180,E1 10437.594,E2 10437.594} C_VEL
LIN {X 0,Y 319.996,Z 849.345,A -85,B 0,C 180,E1 10435.52,E2 10435.52} C_VEL
LIN {X 0,Y 329.439,Z 829.711,A -85,B 0,C 180,E1 10433.815,E2 10433.815} C_VEL
LIN {X 0,Y 338.319,Z 809.008,A -85,B 0,C 180,E1 10432.358,E2 10432.358} C_VEL
LIN {X 0,Y 345.942,Z 788.096,A -85,B 0,C 180,E1 10431.189,E2 10431.189} C_VEL
LIN {X 0,Y 352.903,Z 765.305,A -85,B 0,C 180,E1 10430.19,E2 10430.19} C_VEL
LIN {X 0,Y 357.822,Z 745.241,A -85,B 0,C 180,E1 10429.513,E2 10429.513} C_VEL
LIN {X 0,Y 362.294,Z 721.031,A -85,B 0,C 180,E1 10428.902,E2 10428.902} C_VEL
LIN {X 0,Y 382.885,Z 564.138,A -85,B 0,C 180,E1 10425.752,E2 10425.752} C_VEL
LIN {X 0,Y 382.864,Z 562.47,A -85,B 0,C 180,E1 10424.163,E2 10424.163} C_VEL
LIN {X 0,Y 382.856,Z 564.47,A -85,B 0,C 180,E1 10422.6,E2 10422.6} C_VEL
LIN {X 0,Y 361.144,Z 729.84,A -85,B 0,C 180,E1 10419.291,E2 10419.291} C_VEL
LIN {X 0,Y 356.311,Z 753.701,A -85,B 0,C 180,E1 10418.698,E2 10418.698} C_VEL
LIN {X 0,Y 349.864,Z 777.962,A -85,B 0,C 180,E1 10417.926,E2 10417.926} C_VEL
LIN {X 0,Y 343.538,Z 797.431,A -85,B 0,C 180,E1 10417.103,E2 10417.103} C_VEL
LIN {X 0,Y 334.811,Z 820.288,A -85,B 0,C 180,E1 10415.866,E2 10415.866} C_VEL
LIN {X 0,Y 326.592,Z 839.063,A -85,B 0,C 180,E1 10414.58,E2 10414.58} C_VEL
LIN {X 0,Y 316.429,Z 859.788,A -85,B 0,C 180,E1 10412.815,E2 10412.815} C_VEL
LIN {X 0,Y 305.956,Z 879.144,A -85,B 0,C 180,E1 10410.763,E2 10410.763} C_VEL
LIN {X 0,Y 294.856,Z 897.772,A -85,B 0,C 180,E1 10408.292,E2 10408.292} C_VEL
LIN {X 0,Y 283.817,Z 915.192,A -85,B 0,C 180,E1 10405.447,E2 10405.447} C_VEL
LIN {X 0,Y 273.177,Z 930.918,A -85,B 0,C 180,E1 10402.246,E2 10402.246} C_VEL
LIN {X 0,Y 262.346,Z 946.446,A -85,B 0,C 180,E1 10398.337,E2 10398.337} C_VEL
LIN {X 0,Y 253.223,Z 959.253,A -85,B 0,C 180,E1 10394.344,E2 10394.344} C_VEL
LIN {X 0,Y 244.585,Z 971.444,A -85,B 0,C 180,E1 10389.629,E2 10389.629} C_VEL
LIN {X 0,Y 237.223,Z 982.334,A -85,B 0,C 180,E1 10384.394,E2 10384.394} C_VEL
LIN {X 0,Y 231.602,Z 991.218,A -85,B 0,C 180,E1 10378.922,E2 10378.922} C_VEL
LIN {X 0,Y 227.705,Z 998.518,A -85,B 0,C 180,E1 10373.284,E2 10373.284} C_VEL
LIN {X 0,Y 225.344,Z 1004.039,A -85,B 0,C 180,E1 10367.567,E2 10367.567} C_VEL
LIN {X 0,Y 224.239,Z 1008.095,A -85,B 0,C 180,E1 10361.842,E2 10361.842} C_VEL
LIN {X 0,Y 223.988,Z 1010.225,A -85,B 0,C 180,E1 10356.929,E2 10356.929} C_VEL
LIN {X 0,Y 224.003,Z 1011.184,A -85,B 0,C 180,E1 10352.565,E2 10352.565} C_VEL
LIN {X 0,Y 224.021,Z 1011.215,A -85,B 0,C 180,E1 10348.216,E2 10348.216} C_VEL
LIN {X 0,Y 223.997,Z 1010.17,A -85,B 0,C 180,E1 10343.342,E2 10343.342} C_VEL
LIN {X 0,Y 224.268,Z 1007.495,A -85,B 0,C 180,E1 10337.912,E2 10337.912} C_VEL
LIN {X 0,Y 225.183,Z 1003.85,A -85,B 0,C 180,E1 10332.967,E2 10332.967} C_VEL
LIN {X 0,Y 227.521,Z 997.734,A -85,B 0,C 180,E1 10326.984,E2 10326.984} C_VEL
LIN {X 0,Y 230.885,Z 990.851,A -85,B 0,C 180,E1 10321.842,E2 10321.842} C_VEL
LIN {X 0,Y 236.168,Z 981.414,A -85,B 0,C 180,E1 10316.325,E2 10316.325} C_VEL
LIN {X 0,Y 242.466,Z 971.117,A -85,B 0,C 180,E1 10311.498,E2 10311.498} C_VEL
LIN {X 0,Y 250.16,Z 958.772,A -85,B 0,C 180,E1 10306.895,E2 10306.895} C_VEL
LIN {X 0,Y 258.738,Z 945.156,A -85,B 0,C 180,E1 10302.769,E2 10302.769} C_VEL
LIN {X 0,Y 267.382,Z 930.94,A -85,B 0,C 180,E1 10299.291,E2 10299.291} C_VEL
LIN {X 0,Y 277.46,Z 913.607,A -85,B 0,C 180,E1 10295.837,E2 10295.837} C_VEL
LIN {X 0,Y 286.563,Z 896.977,A -85,B 0,C 180,E1 10293.147,E2 10293.147} C_VEL
LIN {X 0,Y 295.569,Z 879.045,A -85,B 0,C 180,E1 10290.782,E2 10290.782} C_VEL
LIN {X 0,Y 304.367,Z 859.988,A -85,B 0,C 180,E1 10288.719,E2 10288.719} C_VEL
LIN {X 0,Y 312.453,Z 840.177,A -85,B 0,C 180,E1 10286.989,E2 10286.989} C_VEL
LIN {X 0,Y 320.096,Z 819.187,A -85,B 0,C 180,E1 10285.497,E2 10285.497} C_VEL
LIN {X 0,Y 326.44,Z 798.639,A -85,B 0,C 180,E1 10284.342,E2 10284.342} C_VEL
LIN {X 0,Y 332.507,Z 775.383,A -85,B 0,C 180,E1 10283.314,E2 10283.314} C_VEL
LIN {X 0,Y 337.116,Z 753.101,A -85,B 0,C 180,E1 10282.585,E2 10282.585} C_VEL
LIN {X 0,Y 340.676,Z 728.522,A -85,B 0,C 180,E1 10281.964,E2 10281.964} C_VEL
LIN {X 0,Y 356.879,Z 551.206,A -85,B 0,C 180,E1 10278.372,E2 10278.372} C_VEL
LIN {X 0,Y 350.372,Z 540.188,A -85,B 0,C 180,E1 10275.22,E2 10275.22} C_VEL
LIN {X 0,Y 343.851,Z 530.67,A -85,B 0,C 180,E1 10271.659,E2 10271.659} C_VEL
LIN {X 0,Y 340.039,Z 525.38,A -85,B 0,C 180,E1 10269.306,E2 10269.306} C_VEL
LIN {X 0,Y 336.808,Z 520.892,A -85,B 0,C 180,E1 10267.076,E2 10267.076} C_VEL
LIN {X 0,Y 333.373,Z 516.18,A -85,B 0,C 180,E1 10264.386,E2 10264.386} C_VEL
LIN {X 0,Y 329.612,Z 511.08,A -85,B 0,C 180,E1 10260.868,E2 10260.868} C_VEL
LIN {X 0,Y 326.585,Z 507.232,A -85,B 0,C 180,E1 10257.367,E2 10257.367} C_VEL
LIN {X 0,Y 325.726,Z 505.669,A -85,B 0,C 180,E1 10256.127,E2 10256.127} C_VEL
LIN {X 0,Y 322.514,Z 502.22,A -85,B 0,C 180,E1 10250.002,E2 10250.002} C_VEL
LIN {X 0,Y 321.88,Z 500.279,A -85,B 0,C 180,E1 10247.076,E2 10247.076} C_VEL
LIN {X 0,Y 321.59,Z 499.915,A -85,B 0,C 180,E1 10242.26,E2 10242.26} C_VEL
LIN {X 0,Y 322.057,Z 500.715,A -85,B 0,C 180,E1 10239.126,E2 10239.126} C_VEL
LIN {X 0,Y 324.524,Z 504.848,A -85,B 0,C 180,E1 10232.871,E2 10232.871} C_VEL
LIN {X 0,Y 326.069,Z 506.065,A -85,B 0,C 180,E1 10230.618,E2 10230.618} C_VEL
LIN {X 0,Y 328.756,Z 510.26,A -85,B 0,C 180,E1 10227.223,E2 10227.223} C_VEL
LIN {X 0,Y 330.329,Z 511.943,A -85,B 0,C 180,E1 10225.631,E2 10225.631} C_VEL
LIN {X 0,Y 334.574,Z 517.714,A -85,B 0,C 180,E1 10221.894,E2 10221.894} C_VEL
LIN {X 0,Y 338.588,Z 523.3,A -85,B 0,C 180,E1 10218.924,E2 10218.924} C_VEL
LIN {X 0,Y 342.442,Z 528.697,A -85,B 0,C 180,E1 10216.443,E2 10216.443} C_VEL
LIN {X 0,Y 347.959,Z 536.631,A -85,B 0,C 180,E1 10213.304,E2 10213.304} C_VEL
LIN {X 0,Y 355.202,Z 547.618,A -85,B 0,C 180,E1 10209.726,E2 10209.726} C_VEL
LIN {X 0,Y 356.43,Z 549.966,A -85,B 0,C 180,E1 10209.146,E2 10209.146} C_VEL
LIN {X 0,Y 340.835,Z 719.296,A -85,B 0,C 180,E1 10205.723,E2 10205.723} C_VEL
LIN {X 0,Y 337.159,Z 743.175,A -85,B 0,C 180,E1 10205.075,E2 10205.075} C_VEL
LIN {X 0,Y 332.63,Z 765.412,A -85,B 0,C 180,E1 10204.262,E2 10204.262} C_VEL
LIN {X 0,Y 327.08,Z 786.666,A -85,B 0,C 180,E1 10203.242,E2 10203.242} C_VEL
LIN {X 0,Y 320.362,Z 808.482,A -85,B 0,C 180,E1 10201.932,E2 10201.932} C_VEL
LIN {X 0,Y 313.339,Z 827.863,A -85,B 0,C 180,E1 10200.482,E2 10200.482} C_VEL
LIN {X 0,Y 304.582,Z 849.149,A -85,B 0,C 180,E1 10198.524,E2 10198.524} C_VEL
LIN {X 0,Y 296.452,Z 866.771,A -85,B 0,C 180,E1 10196.538,E2 10196.538} C_VEL
LIN {X 0,Y 286.862,Z 885.531,A -85,B 0,C 180,E1 10193.951,E2 10193.951} C_VEL
LIN {X 0,Y 277.556,Z 902.405,A -85,B 0,C 180,E1 10191.108,E2 10191.108} C_VEL
LIN {X 0,Y 268.092,Z 918.214,A -85,B 0,C 180,E1 10187.801,E2 10187.801} C_VEL
LIN {X 0,Y 259.001,Z 932.798,A -85,B 0,C 180,E1 10184.069,E2 10184.069} C_VEL
LIN {X 0,Y 250.846,Z 945.334,A -85,B 0,C 180,E1 10180.094,E2 10180.094} C_VEL
LIN {X 0,Y 243.049,Z 957.269,A -85,B 0,C 180,E1 10175.404,E2 10175.404} C_VEL
LIN {X 0,Y 236.929,Z 966.864,A -85,B 0,C 180,E1 10170.719,E2 10170.719} C_VEL
LIN {X 0,Y 231.624,Z 975.626,A -85,B 0,C 180,E1 10165.289,E2 10165.289} C_VEL
LIN {X 0,Y 227.998,Z 982.479,A -85,B 0,C 180,E1 10159.891,E2 10159.891} C_VEL
LIN {X 0,Y 225.672,Z 987.688,A -85,B 0,C 180,E1 10154.314,E2 10154.314} C_VEL
LIN {X 0,Y 224.507,Z 991.428,A -85,B 0,C 180,E1 10148.848,E2 10148.848} C_VEL
LIN {X 0,Y 224.079,Z 993.606,A -85,B 0,C 180,E1 10143.493,E2 10143.493} C_VEL
LIN {X 0,Y 224.029,Z 994.462,A -85,B 0,C 180,E1 10139.113,E2 10139.113} C_VEL
LIN {X 0,Y 224.057,Z 994.459,A -85,B 0,C 180,E1 10134.534,E2 10134.534} C_VEL
LIN {X 0,Y 224.325,Z 993.217,A -85,B 0,C 180,E1 10129.058,E2 10129.058} C_VEL
LIN {X 0,Y 225.138,Z 990.835,A -85,B 0,C 180,E1 10123.983,E2 10123.983} C_VEL
LIN {X 0,Y 227.044,Z 986.952,A -85,B 0,C 180,E1 10118.375,E2 10118.375} C_VEL
LIN {X 0,Y 230.514,Z 981.105,A -85,B 0,C 180,E1 10112.538,E2 10112.538} C_VEL
LIN {X 0,Y 235.582,Z 973.801,A -85,B 0,C 180,E1 10106.955,E2 10106.955} C_VEL
LIN {X 0,Y 242.036,Z 965.104,A -85,B 0,C 180,E1 10101.827,E2 10101.827} C_VEL
LIN {X 0,Y 250.715,Z 953.823,A -85,B 0,C 180,E1 10096.6,E2 10096.6} C_VEL
LIN {X 0,Y 256.52,Z 946.309,A -85,B 0,C 180,E1 10093.74,E2 10093.74} C_VEL
LIN {X 0,Y 258.704,Z 942.724,A -85,B 0,C 180,E1 10092.292,E2 10092.292} C_VEL
LIN {X 0,Y 262.272,Z 933.362,A -85,B 0,C 180,E1 10088.174,E2 10088.174} C_VEL
LIN {X 0,Y 264.588,Z 929.773,A -85,B 0,C 180,E1 10087.058,E2 10087.058} C_VEL
LIN {X 0,Y 275.527,Z 915.521,A -85,B 0,C 180,E1 10083.619,E2 10083.619} C_VEL
LIN {X 0,Y 286.987,Z 899.4,A -85,B 0,C 180,E1 10080.523,E2 10080.523} C_VEL
LIN {X 0,Y 299.217,Z 880.938,A -85,B 0,C 180,E1 10077.688,E2 10077.688} C_VEL
LIN {X 0,Y 310.591,Z 862.169,A -85,B 0,C 180,E1 10075.384,E2 10075.384} C_VEL
LIN {X 0,Y 321.047,Z 842.723,A -85,B 0,C 180,E1 10073.478,E2 10073.478} C_VEL
LIN {X 0,Y 331.029,Z 821.944,A -85,B 0,C 180,E1 10071.839,E2 10071.839} C_VEL
LIN {X 0,Y 339.29,Z 802.158,A -85,B 0,C 180,E1 10070.587,E2 10070.587} C_VEL
LIN {X 0,Y 347.502,Z 778.968,A -85,B 0,C 180,E1 10069.431,E2 10069.431} C_VEL
LIN {X 0,Y 353.944,Z 756.826,A -85,B 0,C 180,E1 10068.58,E2 10068.58} C_VEL
LIN {X 0,Y 359.142,Z 733.287,A -85,B 0,C 180,E1 10067.913,E2 10067.913} C_VEL
LIN {X 0,Y 363.433,Z 705.743,A -85,B 0,C 180,E1 10067.324,E2 10067.324} C_VEL
LIN {X 0,Y 381.684,Z 571.001,A -85,B 0,C 180,E1 10064.683,E2 10064.683} C_VEL
LIN {X 0,Y 381.724,Z 570.486,A -85,B 0,C 180,E1 10064.193,E2 10064.193} C_VEL
LIN {X 0,Y 381.638,Z 571.354,A -85,B 0,C 180,E1 10063.675,E2 10063.675} C_VEL
LIN {X 0,Y 360.104,Z 729.378,A -85,B 0,C 180,E1 10060.568,E2 10060.568} C_VEL
LIN {X 0,Y 355.146,Z 753.136,A -85,B 0,C 180,E1 10059.995,E2 10059.995} C_VEL
LIN {X 0,Y 348.57,Z 777.281,A -85,B 0,C 180,E1 10059.254,E2 10059.254} C_VEL
LIN {X 0,Y 342.298,Z 796.051,A -85,B 0,C 180,E1 10058.495,E2 10058.495} C_VEL
LIN {X 0,Y 333.293,Z 819.087,A -85,B 0,C 180,E1 10057.298,E2 10057.298} C_VEL
LIN {X 0,Y 324.895,Z 837.672,A -85,B 0,C 180,E1 10056.073,E2 10056.073} C_VEL
LIN {X 0,Y 314.046,Z 859.12,A -85,B 0,C 180,E1 10054.298,E2 10054.298} C_VEL
LIN {X 0,Y 303.597,Z 877.735,A -85,B 0,C 180,E1 10052.371,E2 10052.371} C_VEL
LIN {X 0,Y 291.832,Z 896.803,A -85,B 0,C 180,E1 10049.901,E2 10049.901} C_VEL
LIN {X 0,Y 280.739,Z 913.657,A -85,B 0,C 180,E1 10047.202,E2 10047.202} C_VEL
LIN {X 0,Y 268.822,Z 930.459,A -85,B 0,C 180,E1 10043.821,E2 10043.821} C_VEL
LIN {X 0,Y 256.909,Z 946.639,A -85,B 0,C 180,E1 10039.719,E2 10039.719} C_VEL
LIN {X 0,Y 246.869,Z 959.988,A -85,B 0,C 180,E1 10035.472,E2 10035.472} C_VEL
LIN {X 0,Y 237.811,Z 971.939,A -85,B 0,C 180,E1 10030.675,E2 10030.675} C_VEL
LIN {X 0,Y 230.056,Z 982.663,A -85,B 0,C 180,E1 10025.319,E2 10025.319} C_VEL
LIN {X 0,Y 224.335,Z 991.061,A -85,B 0,C 180,E1 10019.952,E2 10019.952} C_VEL
LIN {X 0,Y 219.953,Z 998.575,A -85,B 0,C 180,E1 10013.871,E2 10013.871} C_VEL
LIN {X 0,Y 217.521,Z 1003.803,A -85,B 0,C 180,E1 10008.221,E2 10008.221} C_VEL
LIN {X 0,Y 216.282,Z 1007.826,A -85,B 0,C 180,E1 10002.285,E2 10002.285} C_VEL
LIN {X 0,Y 215.987,Z 1009.942,A -85,B 0,C 180,E1 9997.187,E2 9997.187} C_VEL
LIN {X 0,Y 215.999,Z 1010.861,A -85,B 0,C 180,E1 9992.926,E2 9992.926} C_VEL
LIN {X 0,Y 216.026,Z 1010.944,A -85,B 0,C 180,E1 9988.652,E2 9988.652} C_VEL
LIN {X 0,Y 216.005,Z 1010.052,A -85,B 0,C 180,E1 9983.896,E2 9983.896} C_VEL
LIN {X 0,Y 216.206,Z 1007.793,A -85,B 0,C 180,E1 9978.537,E2 9978.537} C_VEL
LIN {X 0,Y 217.114,Z 1004.109,A -85,B 0,C 180,E1 9973.142,E2 9973.142} C_VEL
LIN {X 0,Y 219.208,Z 998.865,A -85,B 0,C 180,E1 9967.48,E2 9967.48} C_VEL
LIN {X 0,Y 222.706,Z 991.846,A -85,B 0,C 180,E1 9961.883,E2 9961.883} C_VEL
LIN {X 0,Y 227.779,Z 983.265,A -85,B 0,C 180,E1 9956.43,E2 9956.43} C_VEL
LIN {X 0,Y 234.186,Z 973.108,A -85,B 0,C 180,E1 9951.38,E2 9951.38} C_VEL
LIN {X 0,Y 242.326,Z 960.741,A -85,B 0,C 180,E1 9946.455,E2 9946.455} C_VEL
LIN {X 0,Y 250.728,Z 947.955,A -85,B 0,C 180,E1 9942.371,E2 9942.371} C_VEL
LIN {X 0,Y 260.502,Z 932.659,A -85,B 0,C 180,E1 9938.446,E2 9938.446} C_VEL
LIN {X 0,Y 270.206,Z 916.84,A -85,B 0,C 180,E1 9935.15,E2 9935.15} C_VEL
LIN {X 0,Y 280.108,Z 899.345,A -85,B 0,C 180,E1 9932.236,E2 9932.236} C_VEL
LIN {X 0,Y 290.398,Z 879.711,A -85,B 0,C 180,E1 9929.594,E2 9929.594} C_VEL
LIN {X 0,Y 299.389,Z 860.823,A -85,B 0,C 180,E1 9927.541,E2 9927.541} C_VEL
LIN {X 0,Y 307.981,Z 840.492,A -85,B 0,C 180,E1 9925.76,E2 9925.76} C_VEL
LIN {X 0,Y 315.846,Z 819.516,A -85,B 0,C 180,E1 9924.274,E2 9924.274} C_VEL
LIN {X 0,Y 322.72,Z 797.702,A -85,B 0,C 180,E1 9923.065,E2 9923.065} C_VEL
LIN {X 0,Y 329.066,Z 773.561,A -85,B 0,C 180,E1 9922.032,E2 9922.032} C_VEL
LIN {X 0,Y 333.751,Z 751.048,A -85,B 0,C 180,E1 9921.316,E2 9921.316} C_VEL
LIN {X 0,Y 337.152,Z 727.205,A -85,B 0,C 180,E1 9920.73,E2 9920.73} C_VEL
LIN {X 0,Y 353.222,Z 555.976,A -85,B 0,C 180,E1 9917.269,E2 9917.269} C_VEL
LIN {X 0,Y 347.861,Z 546.849,A -85,B 0,C 180,E1 9914.566,E2 9914.566} C_VEL
LIN {X 0,Y 341.758,Z 537.787,A -85,B 0,C 180,E1 9911.133,E2 9911.133} C_VEL
LIN {X 0,Y 338.169,Z 532.695,A -85,B 0,C 180,E1 9908.844,E2 9908.844} C_VEL
LIN {X 0,Y 334.989,Z 528.241,A -85,B 0,C 180,E1 9906.598,E2 9906.598} C_VEL
LIN {X 0,Y 331.828,Z 523.815,A -85,B 0,C 180,E1 9904.06,E2 9904.06} C_VEL
LIN {X 0,Y 328.309,Z 518.913,A -85,B 0,C 180,E1 9900.697,E2 9900.697} C_VEL
LIN {X 0,Y 325.232,Z 514.96,A -85,B 0,C 180,E1 9897.092,E2 9897.092} C_VEL
LIN {X 0,Y 324.459,Z 513.522,A -85,B 0,C 180,E1 9895.935,E2 9895.935} C_VEL
LIN {X 0,Y 321.327,Z 510.04,A -85,B 0,C 180,E1 9889.783,E2 9889.783} C_VEL
LIN {X 0,Y 320.725,Z 508.16,A -85,B 0,C 180,E1 9886.845,E2 9886.845} C_VEL
LIN {X 0,Y 320.492,Z 507.863,A -85,B 0,C 180,E1 9882.009,E2 9882.009} C_VEL
LIN {X 0,Y 320.923,Z 508.662,A -85,B 0,C 180,E1 9879.156,E2 9879.156} C_VEL
LIN {X 0,Y 323.369,Z 512.766,A -85,B 0,C 180,E1 9872.922,E2 9872.922} C_VEL
LIN {X 0,Y 324.797,Z 513.952,A -85,B 0,C 180,E1 9870.795,E2 9870.795} C_VEL
LIN {X 0,Y 327.554,Z 518.188,A -85,B 0,C 180,E1 9867.296,E2 9867.296} C_VEL
LIN {X 0,Y 329.005,Z 519.869,A -85,B 0,C 180,E1 9865.79,E2 9865.79} C_VEL
LIN {X 0,Y 333.048,Z 525.423,A -85,B 0,C 180,E1 9862.173,E2 9862.173} C_VEL
LIN {X 0,Y 336.945,Z 530.916,A -85,B 0,C 180,E1 9859.244,E2 9859.244} C_VEL
LIN {X 0,Y 340.746,Z 536.353,A -85,B 0,C 180,E1 9856.739,E2 9856.739} C_VEL
LIN {X 0,Y 346.033,Z 544.081,A -85,B 0,C 180,E1 9853.683,E2 9853.683} C_VEL
LIN {X 0,Y 352.811,Z 554.541,A -85,B 0,C 180,E1 9850.25,E2 9850.25} C_VEL
LIN {X 0,Y 337.177,Z 719.621,A -85,B 0,C 180,E1 9846.924,E2 9846.924} C_VEL
LIN {X 0,Y 333.424,Z 743.467,A -85,B 0,C 180,E1 9846.283,E2 9846.283} C_VEL
LIN {X 0,Y 328.871,Z 765.411,A -85,B 0,C 180,E1 9845.492,E2 9845.492} C_VEL
LIN {X 0,Y 323.164,Z 786.838,A -85,B 0,C 180,E1 9844.478,E2 9844.478} C_VEL
LIN {X 0,Y 316.528,Z 808.014,A -85,B 0,C 180,E1 9843.227,E2 9843.227} C_VEL
LIN {X 0,Y 308.972,Z 828.35,A -85,B 0,C 180,E1 9841.719,E2 9841.719} C_VEL
LIN {X 0,Y 299.973,Z 849.609,A -85,B 0,C 180,E1 9839.771,E2 9839.771} C_VEL
LIN {X 0,Y 291.57,Z 867.309,A -85,B 0,C 180,E1 9837.78,E2 9837.78} C_VEL
LIN {X 0,Y 281.723,Z 886.016,A -85,B 0,C 180,E1 9835.2,E2 9835.2} C_VEL
LIN {X 0,Y 272.388,Z 902.426,A -85,B 0,C 180,E1 9832.436,E2 9832.436} C_VEL
LIN {X 0,Y 262.549,Z 918.292,A -85,B 0,C 180,E1 9829.111,E2 9829.111} C_VEL
LIN {X 0,Y 252.887,Z 933.188,A -85,B 0,C 180,E1 9825.262,E2 9825.262} C_VEL
LIN {X 0,Y 244.535,Z 945.501,A -85,B 0,C 180,E1 9821.312,E2 9821.312} C_VEL
LIN {X 0,Y 236.364,Z 957.446,A -85,B 0,C 180,E1 9816.552,E2 9816.552} C_VEL
LIN {X 0,Y 229.861,Z 967.092,A -85,B 0,C 180,E1 9811.738,E2 9811.738} C_VEL
LIN {X 0,Y 224.216,Z 975.87,A -85,B 0,C 180,E1 9806.158,E2 9806.158} C_VEL
LIN {X 0,Y 220.332,Z 982.741,A -85,B 0,C 180,E1 9800.591,E2 9800.591} C_VEL
LIN {X 0,Y 217.826,Z 987.966,A -85,B 0,C 180,E1 9794.826,E2 9794.826} C_VEL
LIN {X 0,Y 216.554,Z 991.711,A -85,B 0,C 180,E1 9789.168,E2 9789.168} C_VEL
LIN {X 0,Y 216.09,Z 993.9,A -85,B 0,C 180,E1 9783.621,E2 9783.621} C_VEL
LIN {X 0,Y 216.034,Z 994.763,A -85,B 0,C 180,E1 9779.08,E2 9779.08} C_VEL
LIN {X 0,Y 216.065,Z 994.767,A -85,B 0,C 180,E1 9774.326,E2 9774.326} C_VEL
LIN {X 0,Y 216.371,Z 993.539,A -85,B 0,C 180,E1 9768.631,E2 9768.631} C_VEL
LIN {X 0,Y 217.312,Z 991.117,A -85,B 0,C 180,E1 9763.28,E2 9763.28} C_VEL
LIN {X 0,Y 219.553,Z 987.059,A -85,B 0,C 180,E1 9757.279,E2 9757.279} C_VEL
LIN {X 0,Y 223.255,Z 981.398,A -85,B 0,C 180,E1 9751.467,E2 9751.467} C_VEL
LIN {X 0,Y 228.871,Z 973.953,A -85,B 0,C 180,E1 9745.627,E2 9745.627} C_VEL
LIN {X 0,Y 235.908,Z 965.161,A -85,B 0,C 180,E1 9740.338,E2 9740.338} C_VEL
LIN {X 0,Y 244.993,Z 954.086,A -85,B 0,C 180,E1 9735.142,E2 9735.142} C_VEL
LIN {X 0,Y 255.035,Z 941.892,A -85,B 0,C 180,E1 9730.619,E2 9730.619} C_VEL
LIN {X 0,Y 264.588,Z 929.773,A -85,B 0,C 180,E1 9727.058,E2 9727.058} C_VEL
LIN {X 0,Y 267.315,Z 925.689,A -85,B 0,C 180,E1 9725.772,E2 9725.772} C_VEL
LIN {X 0,Y 272.548,Z 915.031,A -85,B 0,C 180,E1 9722.033,E2 9722.033} C_VEL
LIN {X 0,Y 275.232,Z 911.014,A -85,B 0,C 180,E1 9721.07,E2 9721.07} C_VEL
LIN {X 0,Y 287.416,Z 894.437,A -85,B 0,C 180,E1 9718.107,E2 9718.107} C_VEL
LIN {X 0,Y 298.365,Z 878.151,A -85,B 0,C 180,E1 9715.773,E2 9715.773} C_VEL
LIN {X 0,Y 310.776,Z 857.902,A -85,B 0,C 180,E1 9713.442,E2 9713.442} C_VEL
LIN {X 0,Y 321.354,Z 838.654,A -85,B 0,C 180,E1 9711.677,E2 9711.677} C_VEL
LIN {X 0,Y 330.757,Z 819.061,A -85,B 0,C 180,E1 9710.238,E2 9710.238} C_VEL
LIN {X 0,Y 339.123,Z 799.415,A -85,B 0,C 180,E1 9709.066,E2 9709.066} C_VEL
LIN {X 0,Y 346.698,Z 778.144,A -85,B 0,C 180,E1 9708.062,E2 9708.062} C_VEL
LIN {X 0,Y 353.354,Z 755.692,A -85,B 0,C 180,E1 9707.238,E2 9707.238} C_VEL
LIN {X 0,Y 358.593,Z 732.233,A -85,B 0,C 180,E1 9706.605,E2 9706.605} C_VEL
LIN {X 0,Y 363.431,Z 701.076,A -85,B 0,C 180,E1 9705.967,E2 9705.967} C_VEL
LIN {X 0,Y 376.323,Z 608.445,A -85,B 0,C 180,E1 9704.19,E2 9704.19} C_VEL
LIN {X 0,Y 359.41,Z 728.796,A -85,B 0,C 180,E1 9701.856,E2 9701.856} C_VEL
LIN {X 0,Y 354.321,Z 752.534,A -85,B 0,C 180,E1 9701.303,E2 9701.303} C_VEL
LIN {X 0,Y 347.7,Z 776.322,A -85,B 0,C 180,E1 9700.604,E2 9700.604} C_VEL
LIN {X 0,Y 341.285,Z 795.021,A -85,B 0,C 180,E1 9699.886,E2 9699.886} C_VEL
LIN {X 0,Y 332.068,Z 818.025,A -85,B 0,C 180,E1 9698.741,E2 9698.741} C_VEL
LIN {X 0,Y 322.645,Z 838.217,A -85,B 0,C 180,E1 9697.448,E2 9697.448} C_VEL
LIN {X 0,Y 311.505,Z 859.328,A -85,B 0,C 180,E1 9695.731,E2 9695.731} C_VEL
LIN {X 0,Y 300.751,Z 877.768,A -85,B 0,C 180,E1 9693.855,E2 9693.855} C_VEL
LIN {X 0,Y 288.96,Z 896.115,A -85,B 0,C 180,E1 9691.516,E2 9691.516} C_VEL
LIN {X 0,Y 277.102,Z 913.382,A -85,B 0,C 180,E1 9688.784,E2 9688.784} C_VEL
LIN {X 0,Y 264.693,Z 930.079,A -85,B 0,C 180,E1 9685.442,E2 9685.442} C_VEL
LIN {X 0,Y 252.195,Z 946.189,A -85,B 0,C 180,E1 9681.362,E2 9681.362} C_VEL
LIN {X 0,Y 241.111,Z 960.134,A -85,B 0,C 180,E1 9676.881,E2 9676.881} C_VEL
LIN {X 0,Y 231.124,Z 972.481,A -85,B 0,C 180,E1 9671.783,E2 9671.783} C_VEL
LIN {X 0,Y 222.626,Z 983.41,A -85,B 0,C 180,E1 9666.047,E2 9666.047} C_VEL
LIN {X 0,Y 216.654,Z 991.656,A -85,B 0,C 180,E1 9660.514,E2 9660.514} C_VEL
LIN {X 0,Y 212.071,Z 998.914,A -85,B 0,C 180,E1 9654.223,E2 9654.223} C_VEL
LIN {X 0,Y 209.54,Z 1004.021,A -85,B 0,C 180,E1 9648.363,E2 9648.363} C_VEL
LIN {X 0,Y 208.27,Z 1007.811,A -85,B 0,C 180,E1 9642.202,E2 9642.202} C_VEL
LIN {X 0,Y 207.989,Z 1009.74,A -85,B 0,C 180,E1 9637.187,E2 9637.187} C_VEL
LIN {X 0,Y 208.007,Z 1010.595,A -85,B 0,C 180,E1 9632.762,E2 9632.762} C_VEL
LIN {X 0,Y 208.032,Z 1010.615,A -85,B 0,C 180,E1 9628.355,E2 9628.355} C_VEL
LIN {X 0,Y 208.006,Z 1009.653,A -85,B 0,C 180,E1 9623.383,E2 9623.383} C_VEL
LIN {X 0,Y 208.274,Z 1007.254,A -85,B 0,C 180,E1 9617.813,E2 9617.813} C_VEL
LIN {X 0,Y 209.274,Z 1003.708,A -85,B 0,C 180,E1 9612.491,E2 9612.491} C_VEL
LIN {X 0,Y 211.689,Z 998.158,A -85,B 0,C 180,E1 9606.39,E2 9606.39} C_VEL
LIN {X 0,Y 215.591,Z 990.991,A -85,B 0,C 180,E1 9600.563,E2 9600.563} C_VEL
LIN {X 0,Y 221.431,Z 981.74,A -85,B 0,C 180,E1 9594.701,E2 9594.701} C_VEL
LIN {X 0,Y 227.957,Z 972.065,A -85,B 0,C 180,E1 9589.862,E2 9589.862} C_VEL
LIN {X 0,Y 236.72,Z 959.371,A -85,B 0,C 180,E1 9584.809,E2 9584.809} C_VEL
LIN {X 0,Y 246.003,Z 945.945,A -85,B 0,C 180,E1 9580.544,E2 9580.544} C_VEL
LIN {X 0,Y 255.851,Z 930.952,A -85,B 0,C 180,E1 9576.774,E2 9576.774} C_VEL
LIN {X 0,Y 266.361,Z 914.208,A -85,B 0,C 180,E1 9573.375,E2 9573.375} C_VEL
LIN {X 0,Y 276.042,Z 897.643,A -85,B 0,C 180,E1 9570.669,E2 9570.669} C_VEL
LIN {X 0,Y 285.934,Z 879.221,A -85,B 0,C 180,E1 9568.228,E2 9568.228} C_VEL
LIN {X 0,Y 295.218,Z 860.19,A -85,B 0,C 180,E1 9566.182,E2 9566.182} C_VEL
LIN {X 0,Y 303.687,Z 840.587,A -85,B 0,C 180,E1 9564.486,E2 9564.486} C_VEL
LIN {X 0,Y 311.735,Z 819.646,A -85,B 0,C 180,E1 9563.015,E2 9563.015} C_VEL
LIN {X 0,Y 318.762,Z 797.917,A -85,B 0,C 180,E1 9561.822,E2 9561.822} C_VEL
LIN {X 0,Y 325.121,Z 774.463,A -85,B 0,C 180,E1 9560.821,E2 9560.821} C_VEL
LIN {X 0,Y 329.876,Z 752.299,A -85,B 0,C 180,E1 9560.119,E2 9560.119} C_VEL
LIN {X 0,Y 333.548,Z 727.859,A -85,B 0,C 180,E1 9559.515,E2 9559.515} C_VEL
LIN {X 0,Y 349.671,Z 560.814,A -85,B 0,C 180,E1 9556.166,E2 9556.166} C_VEL
LIN {X 0,Y 345.369,Z 553.493,A -85,B 0,C 180,E1 9553.903,E2 9553.903} C_VEL
LIN {X 0,Y 339.401,Z 544.522,A -85,B 0,C 180,E1 9550.438,E2 9550.438} C_VEL
LIN {X 0,Y 336.035,Z 539.665,A -85,B 0,C 180,E1 9548.211,E2 9548.211} C_VEL
LIN {X 0,Y 333.304,Z 535.727,A -85,B 0,C 180,E1 9546.199,E2 9546.199} C_VEL
LIN {X 0,Y 330.296,Z 531.45,A -85,B 0,C 180,E1 9543.731,E2 9543.731} C_VEL
LIN {X 0,Y 326.824,Z 526.599,A -85,B 0,C 180,E1 9540.35,E2 9540.35} C_VEL
LIN {X 0,Y 323.826,Z 522.565,A -85,B 0,C 180,E1 9536.725,E2 9536.725} C_VEL
LIN {X 0,Y 323.196,Z 521.376,A -85,B 0,C 180,E1 9535.741,E2 9535.741} C_VEL
LIN {X 0,Y 320.145,Z 517.86,A -85,B 0,C 180,E1 9529.563,E2 9529.563} C_VEL
LIN {X 0,Y 319.598,Z 516.075,A -85,B 0,C 180,E1 9526.798,E2 9526.798} C_VEL
LIN {X 0,Y 319.378,Z 515.792,A -85,B 0,C 180,E1 9521.944,E2 9521.944} C_VEL
LIN {X 0,Y 319.765,Z 516.532,A -85,B 0,C 180,E1 9519.308,E2 9519.308} C_VEL
LIN {X 0,Y 322.156,Z 520.639,A -85,B 0,C 180,E1 9513.055,E2 9513.055} C_VEL
LIN {X 0,Y 323.527,Z 521.836,A -85,B 0,C 180,E1 9510.973,E2 9510.973} C_VEL
LIN {X 0,Y 326.35,Z 526.115,A -85,B 0,C 180,E1 9507.369,E2 9507.369} C_VEL
LIN {X 0,Y 327.595,Z 527.628,A -85,B 0,C 180,E1 9506.045,E2 9506.045} C_VEL
LIN {X 0,Y 331.512,Z 533.109,A -85,B 0,C 180,E1 9502.465,E2 9502.465} C_VEL
LIN {X 0,Y 335.291,Z 538.531,A -85,B 0,C 180,E1 9499.563,E2 9499.563} C_VEL
LIN {X 0,Y 339.023,Z 543.961,A -85,B 0,C 180,E1 9497.056,E2 9497.056} C_VEL
LIN {X 0,Y 344.325,Z 551.903,A -85,B 0,C 180,E1 9493.933,E2 9493.933} C_VEL
LIN {X 0,Y 349.245,Z 559.686,A -85,B 0,C 180,E1 9491.353,E2 9491.353} C_VEL
LIN {X 0,Y 333.661,Z 719.768,A -85,B 0,C 180,E1 9488.153,E2 9488.153} C_VEL
LIN {X 0,Y 329.824,Z 743.647,A -85,B 0,C 180,E1 9487.519,E2 9487.519} C_VEL
LIN {X 0,Y 325.248,Z 765.254,A -85,B 0,C 180,E1 9486.752,E2 9486.752} C_VEL
LIN {X 0,Y 319.283,Z 787.196,A -85,B 0,C 180,E1 9485.728,E2 9485.728} C_VEL
LIN {X 0,Y 312.127,Z 809.351,A -85,B 0,C 180,E1 9484.422,E2 9484.422} C_VEL
LIN {X 0,Y 304.743,Z 828.759,A -85,B 0,C 180,E1 9482.993,E2 9482.993} C_VEL
LIN {X 0,Y 295.508,Z 850.049,A -85,B 0,C 180,E1 9481.056,E2 9481.056} C_VEL
LIN {X 0,Y 286.903,Z 867.691,A -85,B 0,C 180,E1 9479.081,E2 9479.081} C_VEL
LIN {X 0,Y 276.717,Z 886.453,A -85,B 0,C 180,E1 9476.496,E2 9476.496} C_VEL
LIN {X 0,Y 266.777,Z 903.346,A -85,B 0,C 180,E1 9473.635,E2 9473.635} C_VEL
LIN {X 0,Y 256.605,Z 919.164,A -85,B 0,C 180,E1 9470.284,E2 9470.284} C_VEL
LIN {X 0,Y 246.285,Z 934.419,A -85,B 0,C 180,E1 9466.261,E2 9466.261} C_VEL
LIN {X 0,Y 237.466,Z 946.902,A -85,B 0,C 180,E1 9462.146,E2 9462.146} C_VEL
LIN {X 0,Y 228.996,Z 958.647,A -85,B 0,C 180,E1 9457.268,E2 9457.268} C_VEL
LIN {X 0,Y 221.959,Z 968.664,A -85,B 0,C 180,E1 9452.058,E2 9452.058} C_VEL
LIN {X 0,Y 216.373,Z 976.877,A -85,B 0,C 180,E1 9446.514,E2 9446.514} C_VEL
LIN {X 0,Y 212.226,Z 983.81,A -85,B 0,C 180,E1 9440.502,E2 9440.502} C_VEL
LIN {X 0,Y 209.805,Z 988.662,A -85,B 0,C 180,E1 9434.798,E2 9434.798} C_VEL
LIN {X 0,Y 208.484,Z 992.399,A -85,B 0,C 180,E1 9428.617,E2 9428.617} C_VEL
LIN {X 0,Y 208.087,Z 994.291,A -85,B 0,C 180,E1 9423.348,E2 9423.348} C_VEL
LIN {X 0,Y 208.036,Z 995.092,A -85,B 0,C 180,E1 9418.723,E2 9418.723} C_VEL
LIN {X 0,Y 208.077,Z 995.059,A -85,B 0,C 180,E1 9413.761,E2 9413.761} C_VEL
LIN {X 0,Y 208.445,Z 993.811,A -85,B 0,C 180,E1 9408.031,E2 9408.031} C_VEL
LIN {X 0,Y 209.472,Z 991.489,A -85,B 0,C 180,E1 9402.673,E2 9402.673} C_VEL
LIN {X 0,Y 211.938,Z 987.486,A -85,B 0,C 180,E1 9396.473,E2 9396.473} C_VEL
LIN {X 0,Y 216.111,Z 981.678,A -85,B 0,C 180,E1 9390.286,E2 9390.286} C_VEL
LIN {X 0,Y 222.41,Z 973.984,A -85,B 0,C 180,E1 9384.121,E2 9384.121} C_VEL
LIN {X 0,Y 230.107,Z 965.077,A -85,B 0,C 180,E1 9378.678,E2 9378.678} C_VEL
LIN {X 0,Y 239.657,Z 954.14,A -85,B 0,C 180,E1 9373.512,E2 9373.512} C_VEL
LIN {X 0,Y 250.097,Z 942.185,A -85,B 0,C 180,E1 9369.052,E2 9369.052} C_VEL
LIN {X 0,Y 261.05,Z 929,A -85,B 0,C 180,E1 9365.19,E2 9365.19} C_VEL
LIN {X 0,Y 273.739,Z 912.992,A -85,B 0,C 180,E1 9361.466,E2 9361.466} C_VEL
LIN {X 0,Y 275.232,Z 911.014,A -85,B 0,C 180,E1 9361.07,E2 9361.07} C_VEL
LIN {X 0,Y 278.378,Z 906.426,A -85,B 0,C 180,E1 9359.962,E2 9359.962} C_VEL
LIN {X 0,Y 284.919,Z 894.529,A -85,B 0,C 180,E1 9356.641,E2 9356.641} C_VEL
LIN {X 0,Y 287.808,Z 890.104,A -85,B 0,C 180,E1 9355.823,E2 9355.823} C_VEL
LIN {X 0,Y 300.358,Z 871.729,A -85,B 0,C 180,E1 9353.406,E2 9353.406} C_VEL
LIN {X 0,Y 311.451,Z 853.697,A -85,B 0,C 180,E1 9351.508,E2 9351.508} C_VEL
LIN {X 0,Y 322.945,Z 832.67,A -85,B 0,C 180,E1 9349.746,E2 9349.746} C_VEL
LIN {X 0,Y 332.784,Z 812.219,A -85,B 0,C 180,E1 9348.384,E2 9348.384} C_VEL
LIN {X 0,Y 341.345,Z 791.151,A -85,B 0,C 180,E1 9347.28,E2 9347.28} C_VEL
LIN {X 0,Y 349.055,Z 768.692,A -85,B 0,C 180,E1 9346.36,E2 9346.36} C_VEL
LIN {X 0,Y 354.562,Z 748.563,A -85,B 0,C 180,E1 9345.726,E2 9345.726} C_VEL
LIN {X 0,Y 359.635,Z 724.357,A -85,B 0,C 180,E1 9345.152,E2 9345.152} C_VEL
LIN {X 0,Y 366.893,Z 674.573,A -85,B 0,C 180,E1 9344.183,E2 9344.183} C_VEL
LIN {X 0,Y 358.875,Z 729.17,A -85,B 0,C 180,E1 9343.131,E2 9343.131} C_VEL
LIN {X 0,Y 353.591,Z 752.913,A -85,B 0,C 180,E1 9342.596,E2 9342.596} C_VEL
LIN {X 0,Y 347.045,Z 775.762,A -85,B 0,C 180,E1 9341.951,E2 9341.951} C_VEL
LIN {X 0,Y 340.495,Z 794.344,A -85,B 0,C 180,E1 9341.273,E2 9341.273} C_VEL
LIN {X 0,Y 331.077,Z 817.244,A -85,B 0,C 180,E1 9340.183,E2 9340.183} C_VEL
LIN {X 0,Y 321.014,Z 838.154,A -85,B 0,C 180,E1 9338.891,E2 9338.891} C_VEL
LIN {X 0,Y 309.474,Z 859.229,A -85,B 0,C 180,E1 9337.223,E2 9337.223} C_VEL
LIN {X 0,Y 297.745,Z 878.585,A -85,B 0,C 180,E1 9335.288,E2 9335.288} C_VEL
LIN {X 0,Y 285.525,Z 896.73,A -85,B 0,C 180,E1 9332.989,E2 9332.989} C_VEL
LIN {X 0,Y 272.99,Z 914.111,A -85,B 0,C 180,E1 9330.239,E2 9330.239} C_VEL
LIN {X 0,Y 260.795,Z 929.784,A -85,B 0,C 180,E1 9327.108,E2 9327.108} C_VEL
LIN {X 0,Y 247.511,Z 946.035,A -85,B 0,C 180,E1 9322.994,E2 9322.994} C_VEL
LIN {X 0,Y 236.027,Z 959.687,A -85,B 0,C 180,E1 9318.581,E2 9318.581} C_VEL
LIN {X 0,Y 225.838,Z 971.481,A -85,B 0,C 180,E1 9313.69,E2 9313.69} C_VEL
LIN {X 0,Y 216.997,Z 982.096,A -85,B 0,C 180,E1 9308.136,E2 9308.136} C_VEL
LIN {X 0,Y 210.059,Z 990.81,A -85,B 0,C 180,E1 9302.223,E2 9302.223} C_VEL
LIN {X 0,Y 204.607,Z 998.604,A -85,B 0,C 180,E1 9295.308,E2 9295.308} C_VEL
LIN {X 0,Y 201.841,Z 1003.584,A -85,B 0,C 180,E1 9289.391,E2 9289.391} C_VEL
LIN {X 0,Y 200.323,Z 1007.551,A -85,B 0,C 180,E1 9282.694,E2 9282.694} C_VEL
LIN {X 0,Y 199.999,Z 1009.463,A -85,B 0,C 180,E1 9277.476,E2 9277.476} C_VEL
LIN {X 0,Y 200.009,Z 1010.302,A -85,B 0,C 180,E1 9272.873,E2 9272.873} C_VEL
LIN {X 0,Y 200.037,Z 1010.305,A -85,B 0,C 180,E1 9268.289,E2 9268.289} C_VEL
LIN {X 0,Y 200.004,Z 1009.322,A -85,B 0,C 180,E1 9263.117,E2 9263.117} C_VEL
LIN {X 0,Y 200.327,Z 1006.877,A -85,B 0,C 180,E1 9257.322,E2 9257.322} C_VEL
LIN {X 0,Y 201.454,Z 1003.303,A -85,B 0,C 180,E1 9251.788,E2 9251.788} C_VEL
LIN {X 0,Y 204.13,Z 997.634,A -85,B 0,C 180,E1 9245.405,E2 9245.405} C_VEL
LIN {X 0,Y 208.105,Z 990.848,A -85,B 0,C 180,E1 9239.713,E2 9239.713} C_VEL
LIN {X 0,Y 214.296,Z 981.637,A -85,B 0,C 180,E1 9233.672,E2 9233.672} C_VEL
LIN {X 0,Y 221.426,Z 971.643,A -85,B 0,C 180,E1 9228.553,E2 9228.553} C_VEL
LIN {X 0,Y 230.365,Z 959.296,A -85,B 0,C 180,E1 9223.557,E2 9223.557} C_VEL
LIN {X 0,Y 240.048,Z 945.869,A -85,B 0,C 180,E1 9219.232,E2 9219.232} C_VEL
LIN {X 0,Y 250.281,Z 930.912,A -85,B 0,C 180,E1 9215.429,E2 9215.429} C_VEL
LIN {X 0,Y 260.844,Z 914.724,A -85,B 0,C 180,E1 9212.113,E2 9212.113} C_VEL
LIN {X 0,Y 270.812,Z 898.189,A -85,B 0,C 180,E1 9209.401,E2 9209.401} C_VEL
LIN {X 0,Y 281.782,Z 878.332,A -85,B 0,C 180,E1 9206.784,E2 9206.784} C_VEL
LIN {X 0,Y 291.422,Z 859.065,A -85,B 0,C 180,E1 9204.744,E2 9204.744} C_VEL
LIN {X 0,Y 299.971,Z 839.629,A -85,B 0,C 180,E1 9203.097,E2 9203.097} C_VEL
LIN {X 0,Y 308.174,Z 818.663,A -85,B 0,C 180,E1 9201.656,E2 9201.656} C_VEL
LIN {X 0,Y 315.203,Z 797.292,A -85,B 0,C 180,E1 9200.509,E2 9200.509} C_VEL
LIN {X 0,Y 321.778,Z 773.327,A -85,B 0,C 180,E1 9199.515,E2 9199.515} C_VEL
LIN {X 0,Y 326.61,Z 751.03,A -85,B 0,C 180,E1 9198.826,E2 9198.826} C_VEL
LIN {X 0,Y 330.21,Z 727.078,A -85,B 0,C 180,E1 9198.247,E2 9198.247} C_VEL
LIN {X 0,Y 346.185,Z 565.609,A -85,B 0,C 180,E1 9195.023,E2 9195.023} C_VEL
LIN {X 0,Y 341.497,Z 557.814,A -85,B 0,C 180,E1 9192.427,E2 9192.427} C_VEL
LIN {X 0,Y 335.514,Z 548.757,A -85,B 0,C 180,E1 9188.655,E2 9188.655} C_VEL
LIN {X 0,Y 331.492,Z 543.057,A -85,B 0,C 180,E1 9185.712,E2 9185.712} C_VEL
LIN {X 0,Y 328.774,Z 539.083,A -85,B 0,C 180,E1 9183.399,E2 9183.399} C_VEL
LIN {X 0,Y 325.507,Z 534.428,A -85,B 0,C 180,E1 9180.175,E2 9180.175} C_VEL
LIN {X 0,Y 322.49,Z 530.294,A -85,B 0,C 180,E1 9176.444,E2 9176.444} C_VEL
LIN {X 0,Y 321.815,Z 529.159,A -85,B 0,C 180,E1 9175.366,E2 9175.366} C_VEL
LIN {X 0,Y 318.897,Z 525.539,A -85,B 0,C 180,E1 9169.156,E2 9169.156} C_VEL
LIN {X 0,Y 318.461,Z 523.978,A -85,B 0,C 180,E1 9166.699,E2 9166.699} C_VEL
LIN {X 0,Y 318.288,Z 523.739,A -85,B 0,C 180,E1 9161.691,E2 9161.691} C_VEL
LIN {X 0,Y 318.615,Z 524.427,A -85,B 0,C 180,E1 9159.422,E2 9159.422} C_VEL
LIN {X 0,Y 320.97,Z 528.534,A -85,B 0,C 180,E1 9153.147,E2 9153.147} C_VEL
LIN {X 0,Y 322.258,Z 529.716,A -85,B 0,C 180,E1 9151.153,E2 9151.153} C_VEL
LIN {X 0,Y 324.959,Z 533.863,A -85,B 0,C 180,E1 9147.63,E2 9147.63} C_VEL
LIN {X 0,Y 326.192,Z 535.386,A -85,B 0,C 180,E1 9146.302,E2 9146.302} C_VEL
LIN {X 0,Y 330.042,Z 540.894,A -85,B 0,C 180,E1 9142.706,E2 9142.706} C_VEL
LIN {X 0,Y 333.647,Z 546.143,A -85,B 0,C 180,E1 9139.886,E2 9139.886} C_VEL
LIN {X 0,Y 337.34,Z 551.61,A -85,B 0,C 180,E1 9137.358,E2 9137.358} C_VEL
LIN {X 0,Y 342.882,Z 560.113,A -85,B 0,C 180,E1 9134.043,E2 9134.043} C_VEL
LIN {X 0,Y 345.756,Z 564.884,A -85,B 0,C 180,E1 9132.479,E2 9132.479} C_VEL
LIN {X 0,Y 330.225,Z 720.241,A -85,B 0,C 180,E1 9129.397,E2 9129.397} C_VEL
LIN {X 0,Y 326.308,Z 744.049,A -85,B 0,C 180,E1 9128.772,E2 9128.772} C_VEL
LIN {X 0,Y 321.524,Z 766.106,A -85,B 0,C 180,E1 9127.997,E2 9127.997} C_VEL
LIN {X 0,Y 315.459,Z 787.875,A -85,B 0,C 180,E1 9126.991,E2 9126.991} C_VEL
LIN {X 0,Y 308.23,Z 809.696,A -85,B 0,C 180,E1 9125.718,E2 9125.718} C_VEL
LIN {X 0,Y 300.662,Z 829.106,A -85,B 0,C 180,E1 9124.303,E2 9124.303} C_VEL
LIN {X 0,Y 291.182,Z 850.394,A -85,B 0,C 180,E1 9122.382,E2 9122.382} C_VEL
LIN {X 0,Y 282.007,Z 868.71,A -85,B 0,C 180,E1 9120.34,E2 9120.34} C_VEL
LIN {X 0,Y 271.853,Z 886.857,A -85,B 0,C 180,E1 9117.839,E2 9117.839} C_VEL
LIN {X 0,Y 261.895,Z 903.297,A -85,B 0,C 180,E1 9115.066,E2 9115.066} C_VEL
LIN {X 0,Y 251.33,Z 919.173,A -85,B 0,C 180,E1 9111.707,E2 9111.707} C_VEL
LIN {X 0,Y 241.091,Z 933.792,A -85,B 0,C 180,E1 9107.865,E2 9107.865} C_VEL
LIN {X 0,Y 232.271,Z 945.759,A -85,B 0,C 180,E1 9103.942,E2 9103.942} C_VEL
LIN {X 0,Y 222.833,Z 958.312,A -85,B 0,C 180,E1 9098.768,E2 9098.768} C_VEL
LIN {X 0,Y 215.311,Z 968.416,A -85,B 0,C 180,E1 9093.454,E2 9093.454} C_VEL
LIN {X 0,Y 209.316,Z 976.689,A -85,B 0,C 180,E1 9087.803,E2 9087.803} C_VEL
LIN {X 0,Y 204.925,Z 983.534,A -85,B 0,C 180,E1 9081.859,E2 9081.859} C_VEL
LIN {X 0,Y 202.074,Z 988.707,A -85,B 0,C 180,E1 9075.669,E2 9075.669} C_VEL
LIN {X 0,Y 200.617,Z 992.433,A -85,B 0,C 180,E1 9069.552,E2 9069.552} C_VEL
LIN {X 0,Y 200.111,Z 994.475,A -85,B 0,C 180,E1 9063.908,E2 9063.908} C_VEL
LIN {X 0,Y 200.04,Z 995.333,A -85,B 0,C 180,E1 9059.285,E2 9059.285} C_VEL
LIN {X 0,Y 200.074,Z 995.427,A -85,B 0,C 180,E1 9054.548,E2 9054.548} C_VEL
LIN {X 0,Y 200.37,Z 994.552,A -85,B 0,C 180,E1 9048.896,E2 9048.896} C_VEL
LIN {X 0,Y 201.461,Z 992.224,A -85,B 0,C 180,E1 9042.724,E2 9042.724} C_VEL
LIN {X 0,Y 203.734,Z 988.723,A -85,B 0,C 180,E1 9036.781,E2 9036.781} C_VEL
LIN {X 0,Y 208.257,Z 982.926,A -85,B 0,C 180,E1 9029.955,E2 9029.955} C_VEL
LIN {X 0,Y 214.391,Z 975.988,A -85,B 0,C 180,E1 9023.911,E2 9023.911} C_VEL
LIN {X 0,Y 222.231,Z 967.419,A -85,B 0,C 180,E1 9018.302,E2 9018.302} C_VEL
LIN {X 0,Y 232.13,Z 956.911,A -85,B 0,C 180,E1 9012.944,E2 9012.944} C_VEL
LIN {X 0,Y 243.064,Z 945.022,A -85,B 0,C 180,E1 9008.279,E2 9008.279} C_VEL
LIN {X 0,Y 255.592,Z 930.884,A -85,B 0,C 180,E1 9003.962,E2 9003.962} C_VEL
LIN {X 0,Y 267.999,Z 916.181,A -85,B 0,C 180,E1 9000.428,E2 9000.428} C_VEL
LIN {X 0,Y 280.716,Z 899.803,A -85,B 0,C 180,E1 8997.347,E2 8997.347} C_VEL
LIN {X 0,Y 287.808,Z 890.104,A -85,B 0,C 180,E1 8995.823,E2 8995.823} C_VEL
LIN {X 0,Y 291.207,Z 885.005,A -85,B 0,C 180,E1 8994.879,E2 8994.879} C_VEL
LIN {X 0,Y 298.195,Z 872.676,A -85,B 0,C 180,E1 8992.114,E2 8992.114} C_VEL
LIN {X 0,Y 301.631,Z 867.114,A -85,B 0,C 180,E1 8991.309,E2 8991.309} C_VEL
LIN {X 0,Y 313.684,Z 847.59,A -85,B 0,C 180,E1 8989.44,E2 8989.44} C_VEL
LIN {X 0,Y 324.065,Z 828.612,A -85,B 0,C 180,E1 8987.989,E2 8987.989} C_VEL
LIN {X 0,Y 334.263,Z 807.12,A -85,B 0,C 180,E1 8986.684,E2 8986.684} C_VEL
LIN {X 0,Y 342.57,Z 786.749,A -85,B 0,C 180,E1 8985.708,E2 8985.708} C_VEL
LIN {X 0,Y 350.106,Z 764.157,A -85,B 0,C 180,E1 8984.868,E2 8984.868} C_VEL
LIN {X 0,Y 356.03,Z 741.982,A -85,B 0,C 180,E1 8984.25,E2 8984.25} C_VEL
LIN {X 0,Y 356.419,Z 740.127,A -85,B 0,C 180,E1 8984.193,E2 8984.193} C_VEL
LIN {X 0,Y 350.114,Z 764.32,A -85,B 0,C 180,E1 8983.62,E2 8983.62} C_VEL
LIN {X 0,Y 343.034,Z 786.001,A -85,B 0,C 180,E1 8982.956,E2 8982.956} C_VEL
LIN {X 0,Y 334.231,Z 807.918,A -85,B 0,C 180,E1 8982.054,E2 8982.054} C_VEL
LIN {X 0,Y 324.487,Z 828.891,A -85,B 0,C 180,E1 8980.937,E2 8980.937} C_VEL
LIN {X 0,Y 314.558,Z 847.516,A -85,B 0,C 180,E1 8979.675,E2 8979.675} C_VEL
LIN {X 0,Y 302.594,Z 867.718,A -85,B 0,C 180,E1 8977.958,E2 8977.958} C_VEL
LIN {X 0,Y 290.202,Z 886.39,A -85,B 0,C 180,E1 8975.935,E2 8975.935} C_VEL
LIN {X 0,Y 276.044,Z 905.888,A -85,B 0,C 180,E1 8973.241,E2 8973.241} C_VEL
LIN {X 0,Y 262.66,Z 922.989,A -85,B 0,C 180,E1 8970.226,E2 8970.226} C_VEL
LIN {X 0,Y 249.165,Z 938.953,A -85,B 0,C 180,E1 8966.589,E2 8966.589} C_VEL
LIN {X 0,Y 235.678,Z 954.233,A -85,B 0,C 180,E1 8962.109,E2 8962.109} C_VEL
LIN {X 0,Y 223.793,Z 967.399,A -85,B 0,C 180,E1 8957.122,E2 8957.122} C_VEL
LIN {X 0,Y 213.674,Z 978.434,A -85,B 0,C 180,E1 8951.649,E2 8951.649} C_VEL
LIN {X 0,Y 205.191,Z 988.156,A -85,B 0,C 180,E1 8945.449,E2 8945.449} C_VEL
LIN {X 0,Y 199.37,Z 995.366,A -85,B 0,C 180,E1 8939.445,E2 8939.445} C_VEL
LIN {X 0,Y 194.952,Z 1001.834,A -85,B 0,C 180,E1 8932.312,E2 8932.312} C_VEL
LIN {X 0,Y 192.92,Z 1005.793,A -85,B 0,C 180,E1 8926.26,E2 8926.26} C_VEL
LIN {X 0,Y 192.078,Z 1008.715,A -85,B 0,C 180,E1 8919.596,E2 8919.596} C_VEL
LIN {X 0,Y 192.009,Z 1009.886,A -85,B 0,C 180,E1 8914.188,E2 8914.188} C_VEL
LIN {X 0,Y 192.038,Z 1010.066,A -85,B 0,C 180,E1 8909.411,E2 8909.411} C_VEL
LIN {X 0,Y 192.013,Z 1009.397,A -85,B 0,C 180,E1 8904.63,E2 8904.63} C_VEL
LIN {X 0,Y 192.147,Z 1007.638,A -85,B 0,C 180,E1 8899.211,E2 8899.211} C_VEL
LIN {X 0,Y 193.129,Z 1004.18,A -85,B 0,C 180,E1 8892.845,E2 8892.845} C_VEL
LIN {X 0,Y 195.328,Z 999.42,A -85,B 0,C 180,E1 8886.796,E2 8886.796} C_VEL
LIN {X 0,Y 199.697,Z 992.188,A -85,B 0,C 180,E1 8879.964,E2 8879.964} C_VEL
LIN {X 0,Y 205.248,Z 984.215,A -85,B 0,C 180,E1 8874.237,E2 8874.237} C_VEL
LIN {X 0,Y 212.836,Z 974.014,A -85,B 0,C 180,E1 8868.529,E2 8868.529} C_VEL
LIN {X 0,Y 221.686,Z 962.481,A -85,B 0,C 180,E1 8863.447,E2 8863.447} C_VEL
LIN {X 0,Y 231.442,Z 949.459,A -85,B 0,C 180,E1 8858.969,E2 8858.969} C_VEL
LIN {X 0,Y 241.813,Z 935.252,A -85,B 0,C 180,E1 8855.059,E2 8855.059} C_VEL
LIN {X 0,Y 252.489,Z 919.61,A -85,B 0,C 180,E1 8851.65,E2 8851.65} C_VEL
LIN {X 0,Y 264.064,Z 901.431,A -85,B 0,C 180,E1 8848.495,E2 8848.495} C_VEL
LIN {X 0,Y 274.686,Z 883.273,A -85,B 0,C 180,E1 8845.979,E2 8845.979} C_VEL
LIN {X 0,Y 284.756,Z 863.951,A -85,B 0,C 180,E1 8843.856,E2 8843.856} C_VEL
LIN {X 0,Y 294.42,Z 843.29,A -85,B 0,C 180,E1 8842.029,E2 8842.029} C_VEL
LIN {X 0,Y 302.619,Z 823.139,A -85,B 0,C 180,E1 8840.611,E2 8840.611} C_VEL
LIN {X 0,Y 310.48,Z 800.676,A -85,B 0,C 180,E1 8839.361,E2 8839.361} C_VEL
LIN {X 0,Y 316.895,Z 778.797,A -85,B 0,C 180,E1 8838.414,E2 8838.414} C_VEL
LIN {X 0,Y 322.283,Z 755.583,A -85,B 0,C 180,E1 8837.672,E2 8837.672} C_VEL
LIN {X 0,Y 326.348,Z 731.796,A -85,B 0,C 180,E1 8837.074,E2 8837.074} C_VEL
LIN {X 0,Y 338.782,Z 610.411,A -85,B 0,C 180,E1 8834.665,E2 8834.665} C_VEL
LIN {X 0,Y 342.812,Z 570.541,A -85,B 0,C 180,E1 8833.88,E2 8833.88} C_VEL
LIN {X 0,Y 336.841,Z 560.935,A -85,B 0,C 180,E1 8830.345,E2 8830.345} C_VEL
LIN {X 0,Y 332.317,Z 554.257,A -85,B 0,C 180,E1 8827.259,E2 8827.259} C_VEL
LIN {X 0,Y 329.689,Z 550.382,A -85,B 0,C 180,E1 8825.22,E2 8825.22} C_VEL
LIN {X 0,Y 327.227,Z 546.71,A -85,B 0,C 180,E1 8823.065,E2 8823.065} C_VEL
LIN {X 0,Y 324.021,Z 542.106,A -85,B 0,C 180,E1 8819.823,E2 8819.823} C_VEL
LIN {X 0,Y 321.108,Z 537.899,A -85,B 0,C 180,E1 8816.071,E2 8816.071} C_VEL
LIN {X 0,Y 320.563,Z 537.012,A -85,B 0,C 180,E1 8815.169,E2 8815.169} C_VEL
LIN {X 0,Y 317.66,Z 533.212,A -85,B 0,C 180,E1 8808.746,E2 8808.746} C_VEL
LIN {X 0,Y 317.302,Z 531.86,A -85,B 0,C 180,E1 8806.515,E2 8806.515} C_VEL
LIN {X 0,Y 317.204,Z 531.691,A -85,B 0,C 180,E1 8801.436,E2 8801.436} C_VEL
LIN {X 0,Y 317.499,Z 532.459,A -85,B 0,C 180,E1 8799.346,E2 8799.346} C_VEL
LIN {X 0,Y 319.784,Z 536.429,A -85,B 0,C 180,E1 8793.24,E2 8793.24} C_VEL
LIN {X 0,Y 320.993,Z 537.593,A -85,B 0,C 180,E1 8791.334,E2 8791.334} C_VEL
LIN {X 0,Y 323.748,Z 541.788,A -85,B 0,C 180,E1 8787.704,E2 8787.704} C_VEL
LIN {X 0,Y 324.966,Z 543.453,A -85,B 0,C 180,E1 8786.37,E2 8786.37} C_VEL
LIN {X 0,Y 328.472,Z 548.497,A -85,B 0,C 180,E1 8783.045,E2 8783.045} C_VEL
LIN {X 0,Y 332.11,Z 553.907,A -85,B 0,C 180,E1 8780.139,E2 8780.139} C_VEL
LIN {X 0,Y 336.069,Z 559.842,A -85,B 0,C 180,E1 8777.402,E2 8777.402} C_VEL
LIN {X 0,Y 342.109,Z 569.309,A -85,B 0,C 180,E1 8773.789,E2 8773.789} C_VEL
LIN {X 0,Y 342.375,Z 569.994,A -85,B 0,C 180,E1 8773.627,E2 8773.627} C_VEL
LIN {X 0,Y 326.939,Z 720.409,A -85,B 0,C 180,E1 8770.67,E2 8770.67} C_VEL
LIN {X 0,Y 322.936,Z 744.26,A -85,B 0,C 180,E1 8770.054,E2 8770.054} C_VEL
LIN {X 0,Y 318.072,Z 766.23,A -85,B 0,C 180,E1 8769.295,E2 8769.295} C_VEL
LIN {X 0,Y 311.973,Z 787.705,A -85,B 0,C 180,E1 8768.32,E2 8768.32} C_VEL
LIN {X 0,Y 304.444,Z 810.018,A -85,B 0,C 180,E1 8767.041,E2 8767.041} C_VEL
LIN {X 0,Y 296.734,Z 829.386,A -85,B 0,C 180,E1 8765.649,E2 8765.649} C_VEL
LIN {X 0,Y 287.016,Z 850.727,A -85,B 0,C 180,E1 8763.747,E2 8763.747} C_VEL
LIN {X 0,Y 277.588,Z 869.061,A -85,B 0,C 180,E1 8761.72,E2 8761.72} C_VEL
LIN {X 0,Y 267.135,Z 887.204,A -85,B 0,C 180,E1 8759.231,E2 8759.231} C_VEL
LIN {X 0,Y 256.542,Z 904.124,A -85,B 0,C 180,E1 8756.372,E2 8756.372} C_VEL
LIN {X 0,Y 245.63,Z 919.98,A -85,B 0,C 180,E1 8752.995,E2 8752.995} C_VEL
LIN {X 0,Y 234.481,Z 935.243,A -85,B 0,C 180,E1 8748.902,E2 8748.902} C_VEL
LIN {X 0,Y 224.888,Z 947.744,A -85,B 0,C 180,E1 8744.673,E2 8744.673} C_VEL
LIN {X 0,Y 215.991,Z 958.96,A -85,B 0,C 180,E1 8739.855,E2 8739.855} C_VEL
LIN {X 0,Y 208.113,Z 969.047,A -85,B 0,C 180,E1 8734.401,E2 8734.401} C_VEL
LIN {X 0,Y 201.806,Z 977.266,A -85,B 0,C 180,E1 8728.573,E2 8728.573} C_VEL
LIN {X 0,Y 196.992,Z 984.298,A -85,B 0,C 180,E1 8722.116,E2 8722.116} C_VEL
LIN {X 0,Y 194.161,Z 989.173,A -85,B 0,C 180,E1 8715.986,E2 8715.986} C_VEL
LIN {X 0,Y 192.586,Z 992.947,A -85,B 0,C 180,E1 8709.319,E2 8709.319} C_VEL
LIN {X 0,Y 192.111,Z 994.835,A -85,B 0,C 180,E1 8703.736,E2 8703.736} C_VEL
LIN {X 0,Y 192.051,Z 995.656,A -85,B 0,C 180,E1 8698.967,E2 8698.967} C_VEL
LIN {X 0,Y 192.089,Z 995.712,A -85,B 0,C 180,E1 8693.786,E2 8693.786} C_VEL
LIN {X 0,Y 192.534,Z 994.66,A -85,B 0,C 180,E1 8687.514,E2 8687.514} C_VEL
LIN {X 0,Y 193.922,Z 992.181,A -85,B 0,C 180,E1 8681.159,E2 8681.159} C_VEL
LIN {X 0,Y 196.863,Z 988.34,A -85,B 0,C 180,E1 8674.625,E2 8674.625} C_VEL
LIN {X 0,Y 201.737,Z 982.687,A -85,B 0,C 180,E1 8668.078,E2 8668.078} C_VEL
LIN {X 0,Y 208.935,Z 975.245,A -85,B 0,C 180,E1 8661.623,E2 8661.623} C_VEL
LIN {X 0,Y 217.812,Z 966.318,A -85,B 0,C 180,E1 8655.852,E2 8655.852} C_VEL
LIN {X 0,Y 228.765,Z 955.321,A -85,B 0,C 180,E1 8650.429,E2 8650.429} C_VEL
LIN {X 0,Y 240.91,Z 942.912,A -85,B 0,C 180,E1 8645.717,E2 8645.717} C_VEL
LIN {X 0,Y 254.018,Z 928.667,A -85,B 0,C 180,E1 8641.58,E2 8641.58} C_VEL
LIN {X 0,Y 267.47,Z 913.13,A -85,B 0,C 180,E1 8638.073,E2 8638.073} C_VEL
LIN {X 0,Y 280.508,Z 896.981,A -85,B 0,C 180,E1 8635.196,E2 8635.196} C_VEL
LIN {X 0,Y 293.705,Z 878.87,A -85,B 0,C 180,E1 8632.666,E2 8632.666} C_VEL
LIN {X 0,Y 301.631,Z 867.114,A -85,B 0,C 180,E1 8631.309,E2 8631.309} C_VEL
LIN {X 0,Y 305.119,Z 861.526,A -85,B 0,C 180,E1 8630.534,E2 8630.534} C_VEL
LIN {X 0,Y 312.63,Z 848.041,A -85,B 0,C 180,E1 8628.143,E2 8628.143} C_VEL
LIN {X 0,Y 315.996,Z 842.121,A -85,B 0,C 180,E1 8627.475,E2 8627.475} C_VEL
LIN {X 0,Y 326.839,Z 822.057,A -85,B 0,C 180,E1 8626.106,E2 8626.106} C_VEL
LIN {X 0,Y 336.018,Z 802.52,A -85,B 0,C 180,E1 8625.041,E2 8625.041} C_VEL
LIN {X 0,Y 342.63,Z 786.381,A -85,B 0,C 180,E1 8624.301,E2 8624.301} C_VEL
LIN {X 0,Y 333.78,Z 807.793,A -85,B 0,C 180,E1 8623.46,E2 8623.46} C_VEL
LIN {X 0,Y 324.088,Z 828.108,A -85,B 0,C 180,E1 8622.431,E2 8622.431} C_VEL
LIN {X 0,Y 313.691,Z 847.035,A -85,B 0,C 180,E1 8621.21,E2 8621.21} C_VEL
LIN {X 0,Y 301.012,Z 867.719,A -85,B 0,C 180,E1 8619.514,E2 8619.514} C_VEL
LIN {X 0,Y 288.322,Z 886.169,A -85,B 0,C 180,E1 8617.576,E2 8617.576} C_VEL
LIN {X 0,Y 273.694,Z 905.54,A -85,B 0,C 180,E1 8614.966,E2 8614.966} C_VEL
LIN {X 0,Y 259.464,Z 922.945,A -85,B 0,C 180,E1 8611.949,E2 8611.949} C_VEL
LIN {X 0,Y 245.422,Z 938.77,A -85,B 0,C 180,E1 8608.381,E2 8608.381} C_VEL
LIN {X 0,Y 231.302,Z 953.935,A -85,B 0,C 180,E1 8603.943,E2 8603.943} C_VEL
LIN {X 0,Y 218.742,Z 967.03,A -85,B 0,C 180,E1 8598.964,E2 8598.964} C_VEL
LIN {X 0,Y 207.959,Z 978.024,A -85,B 0,C 180,E1 8593.443,E2 8593.443} C_VEL
LIN {X 0,Y 198.446,Z 988.095,A -85,B 0,C 180,E1 8586.847,E2 8586.847} C_VEL
LIN {X 0,Y 191.913,Z 995.57,A -85,B 0,C 180,E1 8580.363,E2 8580.363} C_VEL
LIN {X 0,Y 187.334,Z 1001.643,A -85,B 0,C 180,E1 8573.271,E2 8573.271} C_VEL
LIN {X 0,Y 185.064,Z 1005.569,A -85,B 0,C 180,E1 8566.971,E2 8566.971} C_VEL
LIN {X 0,Y 184.093,Z 1008.442,A -85,B 0,C 180,E1 8560.017,E2 8560.017} C_VEL
LIN {X 0,Y 184.012,Z 1009.594,A -85,B 0,C 180,E1 8554.371,E2 8554.371} C_VEL
LIN {X 0,Y 184.047,Z 1009.771,A -85,B 0,C 180,E1 8549.697,E2 8549.697} C_VEL
LIN {X 0,Y 184.018,Z 1009.129,A -85,B 0,C 180,E1 8544.708,E2 8544.708} C_VEL
LIN {X 0,Y 184.138,Z 1007.506,A -85,B 0,C 180,E1 8539.358,E2 8539.358} C_VEL
LIN {X 0,Y 185.134,Z 1004.189,A -85,B 0,C 180,E1 8532.729,E2 8532.729} C_VEL
LIN {X 0,Y 187.578,Z 999.226,A -85,B 0,C 180,E1 8526.112,E2 8526.112} C_VEL
LIN {X 0,Y 192.128,Z 992.195,A -85,B 0,C 180,E1 8519.167,E2 8519.167} C_VEL
LIN {X 0,Y 197.811,Z 984.482,A -85,B 0,C 180,E1 8513.395,E2 8513.395} C_VEL
LIN {X 0,Y 206.165,Z 973.886,A -85,B 0,C 180,E1 8507.248,E2 8507.248} C_VEL
LIN {X 0,Y 214.951,Z 962.945,A -85,B 0,C 180,E1 8502.316,E2 8502.316} C_VEL
LIN {X 0,Y 225.077,Z 950.055,A -85,B 0,C 180,E1 8497.76,E2 8497.76} C_VEL
LIN {X 0,Y 235.803,Z 935.999,A -85,B 0,C 180,E1 8493.804,E2 8493.804} C_VEL
LIN {X 0,Y 246.809,Z 920.476,A -85,B 0,C 180,E1 8490.373,E2 8490.373} C_VEL
LIN {X 0,Y 258.25,Z 903.216,A -85,B 0,C 180,E1 8487.325,E2 8487.325} C_VEL
LIN {X 0,Y 268.845,Z 885.656,A -85,B 0,C 180,E1 8484.861,E2 8484.861} C_VEL
LIN {X 0,Y 279.901,Z 865.338,A -85,B 0,C 180,E1 8482.589,E2 8482.589} C_VEL
LIN {X 0,Y 289.774,Z 845.038,A -85,B 0,C 180,E1 8480.779,E2 8480.779} C_VEL
LIN {X 0,Y 298.235,Z 824.866,A -85,B 0,C 180,E1 8479.358,E2 8479.358} C_VEL
LIN {X 0,Y 306.351,Z 802.597,A -85,B 0,C 180,E1 8478.111,E2 8478.111} C_VEL
LIN {X 0,Y 312.875,Z 780.991,A -85,B 0,C 180,E1 8477.176,E2 8477.176} C_VEL
LIN {X 0,Y 318.758,Z 756.758,A -85,B 0,C 180,E1 8476.397,E2 8476.397} C_VEL
LIN {X 0,Y 322.991,Z 733.159,A -85,B 0,C 180,E1 8475.805,E2 8475.805} C_VEL
LIN {X 0,Y 330.285,Z 664.431,A -85,B 0,C 180,E1 8474.438,E2 8474.438} C_VEL
LIN {X 0,Y 339.503,Z 575.685,A -85,B 0,C 180,E1 8472.717,E2 8472.717} C_VEL
LIN {X 0,Y 333.798,Z 566.572,A -85,B 0,C 180,E1 8469.134,E2 8469.134} C_VEL
LIN {X 0,Y 329.081,Z 559.279,A -85,B 0,C 180,E1 8465.666,E2 8465.666} C_VEL
LIN {X 0,Y 325.587,Z 554.22,A -85,B 0,C 180,E1 8462.64,E2 8462.64} C_VEL
LIN {X 0,Y 322.547,Z 549.778,A -85,B 0,C 180,E1 8459.467,E2 8459.467} C_VEL
LIN {X 0,Y 319.69,Z 545.377,A -85,B 0,C 180,E1 8455.605,E2 8455.605} C_VEL
LIN {X 0,Y 316.478,Z 541.026,A -85,B 0,C 180,E1 8448.519,E2 8448.519} C_VEL
LIN {X 0,Y 316.139,Z 539.724,A -85,B 0,C 180,E1 8446.278,E2 8446.278} C_VEL
LIN {X 0,Y 316.142,Z 539.698,A -85,B 0,C 180,E1 8440.988,E2 8440.988} C_VEL
LIN {X 0,Y 316.455,Z 540.818,A -85,B 0,C 180,E1 8438.888,E2 8438.888} C_VEL
LIN {X 0,Y 319.077,Z 544.707,A -85,B 0,C 180,E1 8432.571,E2 8432.571} C_VEL
LIN {X 0,Y 319.758,Z 545.534,A -85,B 0,C 180,E1 8431.468,E2 8431.468} C_VEL
LIN {X 0,Y 322.536,Z 549.711,A -85,B 0,C 180,E1 8427.778,E2 8427.778} C_VEL
LIN {X 0,Y 324.276,Z 552.39,A -85,B 0,C 180,E1 8425.863,E2 8425.863} C_VEL
LIN {X 0,Y 326.912,Z 556.099,A -85,B 0,C 180,E1 8423.386,E2 8423.386} C_VEL
LIN {X 0,Y 330.467,Z 561.489,A -85,B 0,C 180,E1 8420.481,E2 8420.481} C_VEL
LIN {X 0,Y 334.958,Z 568.301,A -85,B 0,C 180,E1 8417.343,E2 8417.343} C_VEL
LIN {X 0,Y 339.066,Z 575.208,A -85,B 0,C 180,E1 8414.792,E2 8414.792} C_VEL
LIN {X 0,Y 323.753,Z 720.852,A -85,B 0,C 180,E1 8411.96,E2 8411.96} C_VEL
LIN {X 0,Y 319.678,Z 744.613,A -85,B 0,C 180,E1 8411.356,E2 8411.356} C_VEL
LIN {X 0,Y 314.588,Z 767.059,A -85,B 0,C 180,E1 8410.591,E2 8410.591} C_VEL
LIN {X 0,Y 308.556,Z 787.854,A -85,B 0,C 180,E1 8409.662,E2 8409.662} C_VEL
LIN {X 0,Y 300.896,Z 810.101,A -85,B 0,C 180,E1 8408.41,E2 8408.41} C_VEL
LIN {X 0,Y 292.965,Z 829.584,A -85,B 0,C 180,E1 8407.032,E2 8407.032} C_VEL
LIN {X 0,Y 283.002,Z 850.948,A -85,B 0,C 180,E1 8405.154,E2 8405.154} C_VEL
LIN {X 0,Y 273.324,Z 869.328,A -85,B 0,C 180,E1 8403.146,E2 8403.146} C_VEL
LIN {X 0,Y 262.576,Z 887.521,A -85,B 0,C 180,E1 8400.673,E2 8400.673} C_VEL
LIN {X 0,Y 251.976,Z 904.003,A -85,B 0,C 180,E1 8397.912,E2 8397.912} C_VEL
LIN {X 0,Y 240.81,Z 919.709,A -85,B 0,C 180,E1 8394.589,E2 8394.589} C_VEL
LIN {X 0,Y 229.605,Z 934.554,A -85,B 0,C 180,E1 8390.647,E2 8390.647} C_VEL
LIN {X 0,Y 219.522,Z 947.174,A -85,B 0,C 180,E1 8386.395,E2 8386.395} C_VEL
LIN {X 0,Y 209.666,Z 959.096,A -85,B 0,C 180,E1 8381.267,E2 8381.267} C_VEL
LIN {X 0,Y 201.33,Z 969.206,A -85,B 0,C 180,E1 8375.693,E2 8375.693} C_VEL
LIN {X 0,Y 194.611,Z 977.452,A -85,B 0,C 180,E1 8369.698,E2 8369.698} C_VEL
LIN {X 0,Y 189.627,Z 984.264,A -85,B 0,C 180,E1 8363.331,E2 8363.331} C_VEL
LIN {X 0,Y 186.481,Z 989.201,A -85,B 0,C 180,E1 8356.978,E2 8356.978} C_VEL
LIN {X 0,Y 184.745,Z 992.966,A -85,B 0,C 180,E1 8350.343,E2 8350.343} C_VEL
LIN {X 0,Y 184.137,Z 995.039,A -85,B 0,C 180,E1 8344.245,E2 8344.245} C_VEL
LIN {X 0,Y 184.053,Z 995.934,A -85,B 0,C 180,E1 8339.131,E2 8339.131} C_VEL
LIN {X 0,Y 184.093,Z 996.05,A -85,B 0,C 180,E1 8334.025,E2 8334.025} C_VEL
LIN {X 0,Y 184.453,Z 995.264,A -85,B 0,C 180,E1 8328.175,E2 8328.175} C_VEL
LIN {X 0,Y 185.913,Z 992.93,A -85,B 0,C 180,E1 8321.145,E2 8321.145} C_VEL
LIN {X 0,Y 188.699,Z 989.504,A -85,B 0,C 180,E1 8314.774,E2 8314.774} C_VEL
LIN {X 0,Y 194.29,Z 983.617,A -85,B 0,C 180,E1 8307.26,E2 8307.26} C_VEL
LIN {X 0,Y 201.916,Z 976.369,A -85,B 0,C 180,E1 8300.585,E2 8300.585} C_VEL
LIN {X 0,Y 211.538,Z 967.306,A -85,B 0,C 180,E1 8294.509,E2 8294.509} C_VEL
LIN {X 0,Y 223.696,Z 955.885,A -85,B 0,C 180,E1 8288.742,E2 8288.742} C_VEL
LIN {X 0,Y 236.152,Z 943.875,A -85,B 0,C 180,E1 8284.128,E2 8284.128} C_VEL
LIN {X 0,Y 249.428,Z 930.179,A -85,B 0,C 180,E1 8280.116,E2 8280.116} C_VEL
LIN {X 0,Y 263.861,Z 914.357,A -85,B 0,C 180,E1 8276.525,E2 8276.525} C_VEL
LIN {X 0,Y 275.923,Z 900.052,A -85,B 0,C 180,E1 8273.969,E2 8273.969} C_VEL
LIN {X 0,Y 289.551,Z 882.434,A -85,B 0,C 180,E1 8271.462,E2 8271.462} C_VEL
LIN {X 0,Y 301.175,Z 865.934,A -85,B 0,C 180,E1 8269.586,E2 8269.586} C_VEL
LIN {X 0,Y 313.286,Z 846.739,A -85,B 0,C 180,E1 8267.841,E2 8267.841} C_VEL
LIN {X 0,Y 315.996,Z 842.121,A -85,B 0,C 180,E1 8267.475,E2 8267.475} C_VEL
LIN {X 0,Y 318.238,Z 838.209,A -85,B 0,C 180,E1 8266.989,E2 8266.989} C_VEL
LIN {X 0,Y 323.162,Z 828.993,A -85,B 0,C 180,E1 8265.2,E2 8265.2} C_VEL
LIN {X 0,Y 324.994,Z 825.442,A -85,B 0,C 180,E1 8264.842,E2 8264.842} C_VEL
LIN {X 0,Y 328.751,Z 818.032,A -85,B 0,C 180,E1 8264.412,E2 8264.412} C_VEL
LIN {X 0,Y 317.466,Z 839.395,A -85,B 0,C 180,E1 8263.235,E2 8263.235} C_VEL
LIN {X 0,Y 304.809,Z 860.081,A -85,B 0,C 180,E1 8261.749,E2 8261.749} C_VEL
LIN {X 0,Y 291.435,Z 879.695,A -85,B 0,C 180,E1 8259.936,E2 8259.936} C_VEL
LIN {X 0,Y 277.616,Z 897.909,A -85,B 0,C 180,E1 8257.769,E2 8257.769} C_VEL
LIN {X 0,Y 262.603,Z 915.988,A -85,B 0,C 180,E1 8254.992,E2 8254.992} C_VEL
LIN {X 0,Y 248.387,Z 931.931,A -85,B 0,C 180,E1 8251.84,E2 8251.84} C_VEL
LIN {X 0,Y 233.717,Z 947.152,A -85,B 0,C 180,E1 8247.902,E2 8247.902} C_VEL
LIN {X 0,Y 219.063,Z 961.68,A -85,B 0,C 180,E1 8242.953,E2 8242.953} C_VEL
LIN {X 0,Y 206.417,Z 973.944,A -85,B 0,C 180,E1 8237.423,E2 8237.423} C_VEL
LIN {X 0,Y 195.764,Z 984.163,A -85,B 0,C 180,E1 8231.222,E2 8231.222} C_VEL
LIN {X 0,Y 186.777,Z 993.265,A -85,B 0,C 180,E1 8223.839,E2 8223.839} C_VEL
LIN {X 0,Y 181.225,Z 999.604,A -85,B 0,C 180,E1 8216.907,E2 8216.907} C_VEL
LIN {X 0,Y 177.73,Z 1004.489,A -85,B 0,C 180,E1 8209.393,E2 8209.393} C_VEL
LIN {X 0,Y 176.319,Z 1007.438,A -85,B 0,C 180,E1 8202.785,E2 8202.785} C_VEL
LIN {X 0,Y 176.014,Z 1009.142,A -85,B 0,C 180,E1 8196.204,E2 8196.204} C_VEL
LIN {X 0,Y 176.053,Z 1009.49,A -85,B 0,C 180,E1 8190.334,E2 8190.334} C_VEL
LIN {X 0,Y 176.026,Z 1008.921,A -85,B 0,C 180,E1 8185.121,E2 8185.121} C_VEL
LIN {X 0,Y 176.113,Z 1007.489,A -85,B 0,C 180,E1 8179.872,E2 8179.872} C_VEL
LIN {X 0,Y 176.914,Z 1004.692,A -85,B 0,C 180,E1 8173.595,E2 8173.595} C_VEL
LIN {X 0,Y 179.373,Z 999.823,A -85,B 0,C 180,E1 8166.348,E2 8166.348} C_VEL
LIN {X 0,Y 183.326,Z 993.915,A -85,B 0,C 180,E1 8159.894,E2 8159.894} C_VEL
LIN {X 0,Y 189.731,Z 985.585,A -85,B 0,C 180,E1 8153.087,E2 8153.087} C_VEL
LIN {X 0,Y 197.843,Z 975.873,A -85,B 0,C 180,E1 8146.992,E2 8146.992} C_VEL
LIN {X 0,Y 207.279,Z 964.593,A -85,B 0,C 180,E1 8141.623,E2 8141.623} C_VEL
LIN {X 0,Y 218.232,Z 951.384,A -85,B 0,C 180,E1 8136.713,E2 8136.713} C_VEL
LIN {X 0,Y 229.013,Z 937.766,A -85,B 0,C 180,E1 8132.776,E2 8132.776} C_VEL
LIN {X 0,Y 240.792,Z 921.911,A -85,B 0,C 180,E1 8129.164,E2 8129.164} C_VEL
LIN {X 0,Y 252.285,Z 905.323,A -85,B 0,C 180,E1 8126.164,E2 8126.164} C_VEL
LIN {X 0,Y 263.493,Z 887.398,A -85,B 0,C 180,E1 8123.613,E2 8123.613} C_VEL
LIN {X 0,Y 274.394,Z 868.222,A -85,B 0,C 180,E1 8121.427,E2 8121.427} C_VEL
LIN {X 0,Y 284.035,Z 849.054,A -85,B 0,C 180,E1 8119.691,E2 8119.691} C_VEL
LIN {X 0,Y 293.514,Z 827.618,A -85,B 0,C 180,E1 8118.141,E2 8118.141} C_VEL
LIN {X 0,Y 301.514,Z 806.671,A -85,B 0,C 180,E1 8116.946,E2 8116.946} C_VEL
LIN {X 0,Y 308.542,Z 784.566,A -85,B 0,C 180,E1 8115.968,E2 8115.968} C_VEL
LIN {X 0,Y 314.577,Z 761.549,A -85,B 0,C 180,E1 8115.197,E2 8115.197} C_VEL
LIN {X 0,Y 319.074,Z 738.24,A -85,B 0,C 180,E1 8114.606,E2 8114.606} C_VEL
LIN {X 0,Y 322.936,Z 707.056,A -85,B 0,C 180,E1 8113.957,E2 8113.957} C_VEL
LIN {X 0,Y 336.292,Z 580.979,A -85,B 0,C 180,E1 8111.538,E2 8111.538} C_VEL
LIN {X 0,Y 331.044,Z 572.479,A -85,B 0,C 180,E1 8108.073,E2 8108.073} C_VEL
LIN {X 0,Y 326.749,Z 565.911,A -85,B 0,C 180,E1 8104.739,E2 8104.739} C_VEL
LIN {X 0,Y 324.057,Z 561.841,A -85,B 0,C 180,E1 8102.298,E2 8102.298} C_VEL
LIN {X 0,Y 321.239,Z 557.605,A -85,B 0,C 180,E1 8099.286,E2 8099.286} C_VEL
LIN {X 0,Y 318.38,Z 553.105,A -85,B 0,C 180,E1 8095.316,E2 8095.316} C_VEL
LIN {X 0,Y 315.298,Z 548.839,A -85,B 0,C 180,E1 8088.29,E2 8088.29} C_VEL
LIN {X 0,Y 315.004,Z 547.632,A -85,B 0,C 180,E1 8086.206,E2 8086.206} C_VEL
LIN {X 0,Y 315.014,Z 547.613,A -85,B 0,C 180,E1 8081.039,E2 8081.039} C_VEL
LIN {X 0,Y 315.337,Z 548.868,A -85,B 0,C 180,E1 8078.809,E2 8078.809} C_VEL
LIN {X 0,Y 318.037,Z 552.699,A -85,B 0,C 180,E1 8072.431,E2 8072.431} C_VEL
LIN {X 0,Y 319.265,Z 554.947,A -85,B 0,C 180,E1 8070.445,E2 8070.445} C_VEL
LIN {X 0,Y 322.017,Z 558.651,A -85,B 0,C 180,E1 8067.086,E2 8067.086} C_VEL
LIN {X 0,Y 325.465,Z 563.881,A -85,B 0,C 180,E1 8063.635,E2 8063.635} C_VEL
LIN {X 0,Y 329.018,Z 569.365,A -85,B 0,C 180,E1 8060.682,E2 8060.682} C_VEL
LIN {X 0,Y 333.263,Z 575.979,A -85,B 0,C 180,E1 8057.658,E2 8057.658} C_VEL
LIN {X 0,Y 335.878,Z 580.368,A -85,B 0,C 180,E1 8055.98,E2 8055.98} C_VEL
LIN {X 0,Y 320.7,Z 721.097,A -85,B 0,C 180,E1 8053.275,E2 8053.275} C_VEL
LIN {X 0,Y 316.544,Z 744.858,A -85,B 0,C 180,E1 8052.681,E2 8052.681} C_VEL
LIN {X 0,Y 311.455,Z 766.931,A -85,B 0,C 180,E1 8051.946,E2 8051.946} C_VEL
LIN {X 0,Y 305.296,Z 787.81,A -85,B 0,C 180,E1 8051.036,E2 8051.036} C_VEL
LIN {X 0,Y 297.582,Z 809.896,A -85,B 0,C 180,E1 8049.823,E2 8049.823} C_VEL
LIN {X 0,Y 289.366,Z 829.72,A -85,B 0,C 180,E1 8048.451,E2 8048.451} C_VEL
LIN {X 0,Y 279.164,Z 851.163,A -85,B 0,C 180,E1 8046.6,E2 8046.6} C_VEL
LIN {X 0,Y 269.232,Z 869.565,A -85,B 0,C 180,E1 8044.617,E2 8044.617} C_VEL
LIN {X 0,Y 258.18,Z 887.772,A -85,B 0,C 180,E1 8042.166,E2 8042.166} C_VEL
LIN {X 0,Y 246.917,Z 904.742,A -85,B 0,C 180,E1 8039.331,E2 8039.331} C_VEL
LIN {X 0,Y 235.24,Z 920.65,A -85,B 0,C 180,E1 8035.955,E2 8035.955} C_VEL
LIN {X 0,Y 223.209,Z 935.949,A -85,B 0,C 180,E1 8031.818,E2 8031.818} C_VEL
LIN {X 0,Y 212.786,Z 948.477,A -85,B 0,C 180,E1 8027.493,E2 8027.493} C_VEL
LIN {X 0,Y 203.013,Z 959.698,A -85,B 0,C 180,E1 8022.508,E2 8022.508} C_VEL
LIN {X 0,Y 194.272,Z 969.784,A -85,B 0,C 180,E1 8016.79,E2 8016.79} C_VEL
LIN {X 0,Y 187.197,Z 977.997,A -85,B 0,C 180,E1 8010.604,E2 8010.604} C_VEL
LIN {X 0,Y 181.718,Z 985.005,A -85,B 0,C 180,E1 8003.674,E2 8003.674} C_VEL
LIN {X 0,Y 178.47,Z 989.867,A -85,B 0,C 180,E1 7997.042,E2 7997.042} C_VEL
LIN {X 0,Y 176.655,Z 993.601,A -85,B 0,C 180,E1 7989.794,E2 7989.794} C_VEL
LIN {X 0,Y 176.12,Z 995.474,A -85,B 0,C 180,E1 7983.708,E2 7983.708} C_VEL
LIN {X 0,Y 176.059,Z 996.248,A -85,B 0,C 180,E1 7978.874,E2 7978.874} C_VEL
LIN {X 0,Y 176.104,Z 996.365,A -85,B 0,C 180,E1 7973.731,E2 7973.731} C_VEL
LIN {X 0,Y 176.488,Z 995.651,A -85,B 0,C 180,E1 7967.917,E2 7967.917} C_VEL
LIN {X 0,Y 178.061,Z 993.472,A -85,B 0,C 180,E1 7960.646,E2 7960.646} C_VEL
LIN {X 0,Y 181.297,Z 989.892,A -85,B 0,C 180,E1 7953.604,E2 7953.604} C_VEL
LIN {X 0,Y 187.286,Z 984.177,A -85,B 0,C 180,E1 7945.963,E2 7945.963} C_VEL
LIN {X 0,Y 195.063,Z 977.332,A -85,B 0,C 180,E1 7939.395,E2 7939.395} C_VEL
LIN {X 0,Y 205.085,Z 968.594,A -85,B 0,C 180,E1 7933.247,E2 7933.247} C_VEL
LIN {X 0,Y 216.963,Z 958.234,A -85,B 0,C 180,E1 7927.736,E2 7927.736} C_VEL
LIN {X 0,Y 229.343,Z 946.911,A -85,B 0,C 180,E1 7923.201,E2 7923.201} C_VEL
LIN {X 0,Y 244.158,Z 932.634,A -85,B 0,C 180,E1 7918.828,E2 7918.828} C_VEL
LIN {X 0,Y 258.63,Z 917.736,A -85,B 0,C 180,E1 7915.344,E2 7915.344} C_VEL
LIN {X 0,Y 272.273,Z 902.3,A -85,B 0,C 180,E1 7912.557,E2 7912.557} C_VEL
LIN {X 0,Y 286.225,Z 885.216,A -85,B 0,C 180,E1 7910.116,E2 7910.116} C_VEL
LIN {X 0,Y 298.602,Z 868.367,A -85,B 0,C 180,E1 7908.215,E2 7908.215} C_VEL
LIN {X 0,Y 311.653,Z 848.616,A -85,B 0,C 180,E1 7906.445,E2 7906.445} C_VEL
LIN {X 0,Y 322.851,Z 829.367,A -85,B 0,C 180,E1 7905.083,E2 7905.083} C_VEL
LIN {X 0,Y 324.994,Z 825.442,A -85,B 0,C 180,E1 7904.842,E2 7904.842} C_VEL
LIN {X 0,Y 324.718,Z 825.99,A -85,B 0,C 180,E1 7904.734,E2 7904.734} C_VEL
LIN {X 0,Y 321.562,Z 831.708,A -85,B 0,C 180,E1 7904.618,E2 7904.618} C_VEL
LIN {X 0,Y 313.656,Z 845.183,A -85,B 0,C 180,E1 7904.883,E2 7904.883} C_VEL
LIN {X 0,Y 307.718,Z 854.484,A -85,B 0,C 180,E1 7905.348,E2 7905.348} C_VEL
LIN {X 0,Y 306.862,Z 855.728,A -85,B 0,C 180,E1 7905.446,E2 7905.446} C_VEL
LIN {X 0,Y 294.438,Z 873.377,A -85,B 0,C 180,E1 7907.073,E2 7907.073} C_VEL
LIN {X 0,Y 279.908,Z 891.786,A -85,B 0,C 180,E1 7909.23,E2 7909.23} C_VEL
LIN {X 0,Y 265.246,Z 908.665,A -85,B 0,C 180,E1 7911.765,E2 7911.765} C_VEL
LIN {X 0,Y 249.984,Z 924.492,A -85,B 0,C 180,E1 7914.869,E2 7914.869} C_VEL
LIN {X 0,Y 234.59,Z 939.233,A -85,B 0,C 180,E1 7918.658,E2 7918.658} C_VEL
LIN {X 0,Y 220.287,Z 952.068,A -85,B 0,C 180,E1 7922.99,E2 7922.99} C_VEL
LIN {X 0,Y 206.93,Z 963.232,A -85,B 0,C 180,E1 7928.056,E2 7928.056} C_VEL
LIN {X 0,Y 194.12,Z 973.64,A -85,B 0,C 180,E1 7934.434,E2 7934.434} C_VEL
LIN {X 0,Y 184.346,Z 981.583,A -85,B 0,C 180,E1 7941.092,E2 7941.092} C_VEL
LIN {X 0,Y 176.892,Z 987.703,A -85,B 0,C 180,E1 7948.347,E2 7948.347} C_VEL
LIN {X 0,Y 171.887,Z 992.305,A -85,B 0,C 180,E1 7956.033,E2 7956.033} C_VEL
LIN {X 0,Y 169.281,Z 995.046,A -85,B 0,C 180,E1 7963.396,E2 7963.396} C_VEL
LIN {X 0,Y 168.307,Z 996.45,A -85,B 0,C 180,E1 7970.079,E2 7970.079} C_VEL
LIN {X 0,Y 168.058,Z 996.713,A -85,B 0,C 180,E1 7976.805,E2 7976.805} C_VEL
LIN {X 0,Y 168.098,Z 995.991,A -85,B 0,C 180,E1 7982.733,E2 7982.733} C_VEL
LIN {X 0,Y 168.501,Z 994.387,A -85,B 0,C 180,E1 7988.69,E2 7988.69} C_VEL
LIN {X 0,Y 169.978,Z 991.376,A -85,B 0,C 180,E1 7995.688,E2 7995.688} C_VEL
LIN {X 0,Y 173.239,Z 986.478,A -85,B 0,C 180,E1 8003.084,E2 8003.084} C_VEL
LIN {X 0,Y 178.333,Z 980.315,A -85,B 0,C 180,E1 8009.992,E2 8009.992} C_VEL
LIN {X 0,Y 185.338,Z 972.377,A -85,B 0,C 180,E1 8016.497,E2 8016.497} C_VEL
LIN {X 0,Y 194.132,Z 962.889,A -85,B 0,C 180,E1 8022.484,E2 8022.484} C_VEL
LIN {X 0,Y 203.981,Z 952.043,A -85,B 0,C 180,E1 8027.684,E2 8027.684} C_VEL
LIN {X 0,Y 215.725,Z 938.68,A -85,B 0,C 180,E1 8032.616,E2 8032.616} C_VEL
LIN {X 0,Y 226.759,Z 925.422,A -85,B 0,C 180,E1 8036.437,E2 8036.437} C_VEL
LIN {X 0,Y 238.579,Z 910.058,A -85,B 0,C 180,E1 8039.907,E2 8039.907} C_VEL
LIN {X 0,Y 250.391,Z 893.475,A -85,B 0,C 180,E1 8042.885,E2 8042.885} C_VEL
LIN {X 0,Y 261.609,Z 875.866,A -85,B 0,C 180,E1 8045.374,E2 8045.374} C_VEL
LIN {X 0,Y 273.217,Z 855.565,A -85,B 0,C 180,E1 8047.664,E2 8047.664} C_VEL
LIN {X 0,Y 282.836,Z 836.564,A -85,B 0,C 180,E1 8049.378,E2 8049.378} C_VEL
LIN {X 0,Y 291.846,Z 816.025,A -85,B 0,C 180,E1 8050.863,E2 8050.863} C_VEL
LIN {X 0,Y 299.819,Z 795.085,A -85,B 0,C 180,E1 8052.082,E2 8052.082} C_VEL
LIN {X 0,Y 306.6,Z 773.365,A -85,B 0,C 180,E1 8053.072,E2 8053.072} C_VEL
LIN {X 0,Y 312.551,Z 749.928,A -85,B 0,C 180,E1 8053.898,E2 8053.898} C_VEL
LIN {X 0,Y 316.871,Z 727.288,A -85,B 0,C 180,E1 8054.482,E2 8054.482} C_VEL
LIN {X 0,Y 320.937,Z 694.466,A -85,B 0,C 180,E1 8055.141,E2 8055.141} C_VEL
LIN {X 0,Y 332.697,Z 585.565,A -85,B 0,C 180,E1 8057.218,E2 8057.218} C_VEL
LIN {X 0,Y 327.89,Z 577.724,A -85,B 0,C 180,E1 8060.634,E2 8060.634} C_VEL
LIN {X 0,Y 324.644,Z 572.69,A -85,B 0,C 180,E1 8063.309,E2 8063.309} C_VEL
LIN {X 0,Y 322.398,Z 569.238,A -85,B 0,C 180,E1 8065.42,E2 8065.42} C_VEL
LIN {X 0,Y 319.771,Z 565.209,A -85,B 0,C 180,E1 8068.311,E2 8068.311} C_VEL
LIN {X 0,Y 316.824,Z 560.578,A -85,B 0,C 180,E1 8072.563,E2 8072.563} C_VEL
LIN {X 0,Y 314.175,Z 556.77,A -85,B 0,C 180,E1 8078.922,E2 8078.922} C_VEL
LIN {X 0,Y 313.884,Z 555.53,A -85,B 0,C 180,E1 8081.078,E2 8081.078} C_VEL
LIN {X 0,Y 313.885,Z 555.579,A -85,B 0,C 180,E1 8086.273,E2 8086.273} C_VEL
LIN {X 0,Y 316.089,Z 560.016,A -85,B 0,C 180,E1 8093.461,E2 8093.461} C_VEL
LIN {X 0,Y 317.165,Z 561.083,A -85,B 0,C 180,E1 8095.207,E2 8095.207} C_VEL
LIN {X 0,Y 320.093,Z 565.588,A -85,B 0,C 180,E1 8099.284,E2 8099.284} C_VEL
LIN {X 0,Y 323.934,Z 571.535,A -85,B 0,C 180,E1 8103.273,E2 8103.273} C_VEL
LIN {X 0,Y 327.397,Z 576.992,A -85,B 0,C 180,E1 8106.223,E2 8106.223} C_VEL
LIN {X 0,Y 331.593,Z 583.656,A -85,B 0,C 180,E1 8109.283,E2 8109.283} C_VEL
LIN {X 0,Y 333.127,Z 586.58,A -85,B 0,C 180,E1 8110.352,E2 8110.352} C_VEL
LIN {X 0,Y 317.281,Z 730.826,A -85,B 0,C 180,E1 8113.096,E2 8113.096} C_VEL
LIN {X 0,Y 313.002,Z 754.701,A -85,B 0,C 180,E1 8113.663,E2 8113.663} C_VEL
LIN {X 0,Y 307.492,Z 777.425,A -85,B 0,C 180,E1 8114.333,E2 8114.333} C_VEL
LIN {X 0,Y 300.926,Z 798.765,A -85,B 0,C 180,E1 8115.184,E2 8115.184} C_VEL
LIN {X 0,Y 292.73,Z 821.129,A -85,B 0,C 180,E1 8116.328,E2 8116.328} C_VEL
LIN {X 0,Y 284.253,Z 840.818,A -85,B 0,C 180,E1 8117.615,E2 8117.615} C_VEL
LIN {X 0,Y 273.885,Z 861.817,A -85,B 0,C 180,E1 8119.341,E2 8119.341} C_VEL
LIN {X 0,Y 263.4,Z 880.665,A -85,B 0,C 180,E1 8121.286,E2 8121.286} C_VEL
LIN {X 0,Y 252.093,Z 898.74,A -85,B 0,C 180,E1 8123.643,E2 8123.643} C_VEL
LIN {X 0,Y 240.452,Z 915.799,A -85,B 0,C 180,E1 8126.418,E2 8126.418} C_VEL
LIN {X 0,Y 228.847,Z 931.222,A -85,B 0,C 180,E1 8129.622,E2 8129.622} C_VEL
LIN {X 0,Y 216.376,Z 946.748,A -85,B 0,C 180,E1 8133.735,E2 8133.735} C_VEL
LIN {X 0,Y 205.63,Z 959.389,A -85,B 0,C 180,E1 8138.042,E2 8138.042} C_VEL
LIN {X 0,Y 194.834,Z 971.624,A -85,B 0,C 180,E1 8143.444,E2 8143.444} C_VEL
LIN {X 0,Y 185.761,Z 981.969,A -85,B 0,C 180,E1 8149.374,E2 8149.374} C_VEL
LIN {X 0,Y 178.405,Z 990.516,A -85,B 0,C 180,E1 8155.925,E2 8155.925} C_VEL
LIN {X 0,Y 172.909,Z 997.728,A -85,B 0,C 180,E1 8163.2,E2 8163.2} C_VEL
LIN {X 0,Y 169.845,Z 1002.659,A -85,B 0,C 180,E1 8170.046,E2 8170.046} C_VEL
LIN {X 0,Y 168.314,Z 1006.409,A -85,B 0,C 180,E1 8177.313,E2 8177.313} C_VEL
LIN {X 0,Y 168.033,Z 1008.375,A -85,B 0,C 180,E1 8183.861,E2 8183.861} C_VEL
LIN {X 0,Y 168.057,Z 1009.103,A -85,B 0,C 180,E1 8188.986,E2 8188.986} C_VEL
LIN {X 0,Y 168.021,Z 1009.074,A -85,B 0,C 180,E1 8194.104,E2 8194.104} C_VEL
LIN {X 0,Y 168.081,Z 1008.227,A -85,B 0,C 180,E1 8199.597,E2 8199.597} C_VEL
LIN {X 0,Y 168.85,Z 1006.187,A -85,B 0,C 180,E1 8206.168,E2 8206.168} C_VEL
LIN {X 0,Y 171.549,Z 1002.182,A -85,B 0,C 180,E1 8214.087,E2 8214.087} C_VEL
LIN {X 0,Y 176.33,Z 996.805,A -85,B 0,C 180,E1 8221.453,E2 8221.453} C_VEL
LIN {X 0,Y 184.277,Z 989.054,A -85,B 0,C 180,E1 8229.115,E2 8229.115} C_VEL
LIN {X 0,Y 194.214,Z 980.102,A -85,B 0,C 180,E1 8235.702,E2 8235.702} C_VEL
LIN {X 0,Y 206.481,Z 969.012,A -85,B 0,C 180,E1 8241.698,E2 8241.698} C_VEL
LIN {X 0,Y 221.347,Z 955.414,A -85,B 0,C 180,E1 8247.177,E2 8247.177} C_VEL
LIN {X 0,Y 235.945,Z 941.518,A -85,B 0,C 180,E1 8251.39,E2 8251.39} C_VEL
LIN {X 0,Y 250.734,Z 926.362,A -85,B 0,C 180,E1 8254.862,E2 8254.862} C_VEL
LIN {X 0,Y 266.141,Z 909.515,A -85,B 0,C 180,E1 8257.84,E2 8257.84} C_VEL
LIN {X 0,Y 279.32,Z 893.796,A -85,B 0,C 180,E1 8260.003,E2 8260.003} C_VEL
LIN {X 0,Y 293.799,Z 874.967,A -85,B 0,C 180,E1 8262.036,E2 8262.036} C_VEL
LIN {X 0,Y 306.031,Z 857.258,A -85,B 0,C 180,E1 8263.53,E2 8263.53} C_VEL
LIN {X 0,Y 314.808,Z 843.323,A -85,B 0,C 180,E1 8264.5,E2 8264.5} C_VEL
LIN {X 0,Y 306.862,Z 855.728,A -85,B 0,C 180,E1 8265.446,E2 8265.446} C_VEL
LIN {X 0,Y 304.838,Z 858.707,A -85,B 0,C 180,E1 8265.527,E2 8265.527} C_VEL
LIN {X 0,Y 301.997,Z 862.862,A -85,B 0,C 180,E1 8265.272,E2 8265.272} C_VEL
LIN {X 0,Y 294.387,Z 873.349,A -85,B 0,C 180,E1 8263.824,E2 8263.824} C_VEL
LIN {X 0,Y 293.951,Z 873.948,A -85,B 0,C 180,E1 8263.768,E2 8263.768} C_VEL
LIN {X 0,Y 278.891,Z 892.985,A -85,B 0,C 180,E1 8261.827,E2 8261.827} C_VEL
LIN {X 0,Y 264.503,Z 909.556,A -85,B 0,C 180,E1 8259.642,E2 8259.642} C_VEL
LIN {X 0,Y 248.706,Z 926.12,A -85,B 0,C 180,E1 8256.798,E2 8256.798} C_VEL
LIN {X 0,Y 233.547,Z 940.978,A -85,B 0,C 180,E1 8253.489,E2 8253.489} C_VEL
LIN {X 0,Y 217.673,Z 955.337,A -85,B 0,C 180,E1 8249.21,E2 8249.21} C_VEL
LIN {X 0,Y 202.647,Z 968.303,A -85,B 0,C 180,E1 8244.025,E2 8244.025} C_VEL
LIN {X 0,Y 189.528,Z 979.367,A -85,B 0,C 180,E1 8238.07,E2 8238.07} C_VEL
LIN {X 0,Y 178.606,Z 988.442,A -85,B 0,C 180,E1 8231.353,E2 8231.353} C_VEL
LIN {X 0,Y 169.879,Z 996.172,A -85,B 0,C 180,E1 8223.6,E2 8223.6} C_VEL
LIN {X 0,Y 164.405,Z 1001.59,A -85,B 0,C 180,E1 8215.978,E2 8215.978} C_VEL
LIN {X 0,Y 161.079,Z 1005.828,A -85,B 0,C 180,E1 8207.344,E2 8207.344} C_VEL
LIN {X 0,Y 160.113,Z 1007.885,A -85,B 0,C 180,E1 8200.443,E2 8200.443} C_VEL
LIN {X 0,Y 160.024,Z 1008.786,A -85,B 0,C 180,E1 8194.309,E2 8194.309} C_VEL
LIN {X 0,Y 160.064,Z 1008.786,A -85,B 0,C 180,E1 8188.936,E2 8188.936} C_VEL
LIN {X 0,Y 160.029,Z 1007.957,A -85,B 0,C 180,E1 8183.192,E2 8183.192} C_VEL
LIN {X 0,Y 160.483,Z 1005.698,A -85,B 0,C 180,E1 8175.948,E2 8175.948} C_VEL
LIN {X 0,Y 162.244,Z 1001.985,A -85,B 0,C 180,E1 8168.689,E2 8168.689} C_VEL
LIN {X 0,Y 165.981,Z 996.675,A -85,B 0,C 180,E1 8161.201,E2 8161.201} C_VEL
LIN {X 0,Y 171.985,Z 989.421,A -85,B 0,C 180,E1 8153.908,E2 8153.908} C_VEL
LIN {X 0,Y 180.318,Z 980.311,A -85,B 0,C 180,E1 8147.011,E2 8147.011} C_VEL
LIN {X 0,Y 189.373,Z 970.589,A -85,B 0,C 180,E1 8141.447,E2 8141.447} C_VEL
LIN {X 0,Y 201.119,Z 957.836,A -85,B 0,C 180,E1 8135.886,E2 8135.886} C_VEL
LIN {X 0,Y 213.106,Z 944.297,A -85,B 0,C 180,E1 8131.377,E2 8131.377} C_VEL
LIN {X 0,Y 225.499,Z 929.182,A -85,B 0,C 180,E1 8127.545,E2 8127.545} C_VEL
LIN {X 0,Y 238.392,Z 912.27,A -85,B 0,C 180,E1 8124.204,E2 8124.204} C_VEL
LIN {X 0,Y 249.614,Z 896.127,A -85,B 0,C 180,E1 8121.695,E2 8121.695} C_VEL
LIN {X 0,Y 261.678,Z 876.882,A -85,B 0,C 180,E1 8119.328,E2 8119.328} C_VEL
LIN {X 0,Y 272.473,Z 857.651,A -85,B 0,C 180,E1 8117.454,E2 8117.454} C_VEL
LIN {X 0,Y 282.679,Z 836.683,A -85,B 0,C 180,E1 8115.854,E2 8115.854} C_VEL
LIN {X 0,Y 291.954,Z 814.762,A -85,B 0,C 180,E1 8114.539,E2 8114.539} C_VEL
LIN {X 0,Y 299.29,Z 794.292,A -85,B 0,C 180,E1 8113.58,E2 8113.58} C_VEL
LIN {X 0,Y 306.268,Z 770.647,A -85,B 0,C 180,E1 8112.735,E2 8112.735} C_VEL
LIN {X 0,Y 311.665,Z 747.441,A -85,B 0,C 180,E1 8112.107,E2 8112.107} C_VEL
LIN {X 0,Y 315.413,Z 723.606,A -85,B 0,C 180,E1 8111.59,E2 8111.59} C_VEL
LIN {X 0,Y 330.096,Z 591.675,A -85,B 0,C 180,E1 8109.101,E2 8109.101} C_VEL
LIN {X 0,Y 326.006,Z 584.959,A -85,B 0,C 180,E1 8106.073,E2 8106.073} C_VEL
LIN {X 0,Y 321.755,Z 577.996,A -85,B 0,C 180,E1 8102.315,E2 8102.315} C_VEL
LIN {X 0,Y 318.332,Z 572.931,A -85,B 0,C 180,E1 8098.56,E2 8098.56} C_VEL
LIN {X 0,Y 315.485,Z 568.398,A -85,B 0,C 180,E1 8094.361,E2 8094.361} C_VEL
LIN {X 0,Y 312.945,Z 564.464,A -85,B 0,C 180,E1 8087.826,E2 8087.826} C_VEL
LIN {X 0,Y 312.709,Z 563.414,A -85,B 0,C 180,E1 8085.936,E2 8085.936} C_VEL
LIN {X 0,Y 312.766,Z 563.479,A -85,B 0,C 180,E1 8080.969,E2 8080.969} C_VEL
LIN {X 0,Y 315.146,Z 568.108,A -85,B 0,C 180,E1 8073.426,E2 8073.426} C_VEL
LIN {X 0,Y 315.957,Z 569.072,A -85,B 0,C 180,E1 8072.072,E2 8072.072} C_VEL
LIN {X 0,Y 319.299,Z 574.307,A -85,B 0,C 180,E1 8067.517,E2 8067.517} C_VEL
LIN {X 0,Y 322.476,Z 579.259,A -85,B 0,C 180,E1 8064.235,E2 8064.235} C_VEL
LIN {X 0,Y 325.915,Z 584.771,A -85,B 0,C 180,E1 8061.255,E2 8061.255} C_VEL
LIN {X 0,Y 329.722,Z 591.159,A -85,B 0,C 180,E1 8058.405,E2 8058.405} C_VEL
LIN {X 0,Y 314.988,Z 721.637,A -85,B 0,C 180,E1 8055.969,E2 8055.969} C_VEL
LIN {X 0,Y 310.653,Z 745.51,A -85,B 0,C 180,E1 8055.398,E2 8055.398} C_VEL
LIN {X 0,Y 305.291,Z 767.845,A -85,B 0,C 180,E1 8054.686,E2 8054.686} C_VEL
LIN {X 0,Y 298.895,Z 788.711,A -85,B 0,C 180,E1 8053.816,E2 8053.816} C_VEL
LIN {X 0,Y 290.754,Z 811.042,A -85,B 0,C 180,E1 8052.636,E2 8052.636} C_VEL
LIN {X 0,Y 282.299,Z 830.615,A -85,B 0,C 180,E1 8051.333,E2 8051.333} C_VEL
LIN {X 0,Y 271.627,Z 852.057,A -85,B 0,C 180,E1 8049.546,E2 8049.546} C_VEL
LIN {X 0,Y 260.826,Z 871.139,A -85,B 0,C 180,E1 8047.546,E2 8047.546} C_VEL
LIN {X 0,Y 249.188,Z 889.237,A -85,B 0,C 180,E1 8045.146,E2 8045.146} C_VEL
LIN {X 0,Y 237.267,Z 906.111,A -85,B 0,C 180,E1 8042.348,E2 8042.348} C_VEL
LIN {X 0,Y 225.522,Z 921.161,A -85,B 0,C 180,E1 8039.18,E2 8039.18} C_VEL
LIN {X 0,Y 212.561,Z 936.524,A -85,B 0,C 180,E1 8035.037,E2 8035.037} C_VEL
LIN {X 0,Y 201.244,Z 949.093,A -85,B 0,C 180,E1 8030.647,E2 8030.647} C_VEL
LIN {X 0,Y 190.516,Z 960.339,A -85,B 0,C 180,E1 8025.516,E2 8025.516} C_VEL
LIN {X 0,Y 180.81,Z 970.438,A -85,B 0,C 180,E1 8019.541,E2 8019.541} C_VEL
LIN {X 0,Y 172.853,Z 978.662,A -85,B 0,C 180,E1 8012.975,E2 8012.975} C_VEL
LIN {X 0,Y 166.517,Z 985.759,A -85,B 0,C 180,E1 8005.393,E2 8005.393} C_VEL
LIN {X 0,Y 162.843,Z 990.524,A -85,B 0,C 180,E1 7998.301,E2 7998.301} C_VEL
LIN {X 0,Y 160.738,Z 994.235,A -85,B 0,C 180,E1 7990.363,E2 7990.363} C_VEL
LIN {X 0,Y 160.142,Z 996.028,A -85,B 0,C 180,E1 7984.039,E2 7984.039} C_VEL
LIN {X 0,Y 160.068,Z 996.836,A -85,B 0,C 180,E1 7978.761,E2 7978.761} C_VEL
LIN {X 0,Y 160.133,Z 996.998,A -85,B 0,C 180,E1 7973.058,E2 7973.058} C_VEL
LIN {X 0,Y 160.582,Z 996.424,A -85,B 0,C 180,E1 7967.248,E2 7967.248} C_VEL
LIN {X 0,Y 162.35,Z 994.616,A -85,B 0,C 180,E1 7959.649,E2 7959.649} C_VEL
LIN {X 0,Y 166.344,Z 991.024,A -85,B 0,C 180,E1 7951.531,E2 7951.531} C_VEL
LIN {X 0,Y 173.168,Z 985.728,A -85,B 0,C 180,E1 7943.479,E2 7943.479} C_VEL
LIN {X 0,Y 182.44,Z 978.77,A -85,B 0,C 180,E1 7936.232,E2 7936.232} C_VEL
LIN {X 0,Y 194.63,Z 969.645,A -85,B 0,C 180,E1 7929.444,E2 7929.444} C_VEL
LIN {X 0,Y 208.086,Z 959.346,A -85,B 0,C 180,E1 7923.858,E2 7923.858} C_VEL
LIN {X 0,Y 223.174,Z 946.986,A -85,B 0,C 180,E1 7918.974,E2 7918.974} C_VEL
LIN {X 0,Y 238.923,Z 933.182,A -85,B 0,C 180,E1 7914.917,E2 7914.917} C_VEL
LIN {X 0,Y 254.718,Z 918.246,A -85,B 0,C 180,E1 7911.593,E2 7911.593} C_VEL
LIN {X 0,Y 270.051,Z 902.161,A -85,B 0,C 180,E1 7908.878,E2 7908.878} C_VEL
LIN {X 0,Y 286.179,Z 883.502,A -85,B 0,C 180,E1 7906.463,E2 7906.463} C_VEL
LIN {X 0,Y 300.313,Z 865.281,A -85,B 0,C 180,E1 7904.642,E2 7904.642} C_VEL
LIN {X 0,Y 300.834,Z 864.582,A -85,B 0,C 180,E1 7904.559,E2 7904.559} C_VEL
LIN {X 0,Y 293.951,Z 873.948,A -85,B 0,C 180,E1 7903.768,E2 7903.768} C_VEL
LIN {X 0,Y 289.38,Z 879.983,A -85,B 0,C 180,E1 7903.42,E2 7903.42} C_VEL
LIN {X 0,Y 276.441,Z 895.29,A -85,B 0,C 180,E1 7903.101,E2 7903.101} C_VEL
LIN {X 0,Y 271.407,Z 900.775,A -85,B 0,C 180,E1 7902.66,E2 7902.66} C_VEL
LIN {X 0,Y 255.932,Z 917.121,A -85,B 0,C 180,E1 7900.321,E2 7900.321} C_VEL
LIN {X 0,Y 238.693,Z 933.847,A -85,B 0,C 180,E1 7897.166,E2 7897.166} C_VEL
LIN {X 0,Y 223.908,Z 947.135,A -85,B 0,C 180,E1 7893.851,E2 7893.851} C_VEL
LIN {X 0,Y 207.629,Z 960.823,A -85,B 0,C 180,E1 7889.307,E2 7889.307} C_VEL
LIN {X 0,Y 192.856,Z 972.714,A -85,B 0,C 180,E1 7883.987,E2 7883.987} C_VEL
LIN {X 0,Y 179.625,Z 982.908,A -85,B 0,C 180,E1 7877.661,E2 7877.661} C_VEL
LIN {X 0,Y 168.024,Z 991.985,A -85,B 0,C 180,E1 7869.859,E2 7869.859} C_VEL
LIN {X 0,Y 160.095,Z 998.627,A -85,B 0,C 180,E1 7861.859,E2 7861.859} C_VEL
LIN {X 0,Y 154.932,Z 1003.562,A -85,B 0,C 180,E1 7853.192,E2 7853.192} C_VEL
LIN {X 0,Y 152.706,Z 1006.497,A -85,B 0,C 180,E1 7845.582,E2 7845.582} C_VEL
LIN {X 0,Y 152.017,Z 1008.233,A -85,B 0,C 180,E1 7837.569,E2 7837.569} C_VEL
LIN {X 0,Y 152.067,Z 1008.584,A -85,B 0,C 180,E1 7831.517,E2 7831.517} C_VEL
LIN {X 0,Y 152.043,Z 1008.143,A -85,B 0,C 180,E1 7825.862,E2 7825.862} C_VEL
LIN {X 0,Y 152.123,Z 1006.812,A -85,B 0,C 180,E1 7819.788,E2 7819.788} C_VEL
LIN {X 0,Y 152.997,Z 1004.271,A -85,B 0,C 180,E1 7812.908,E2 7812.908} C_VEL
LIN {X 0,Y 155.786,Z 999.843,A -85,B 0,C 180,E1 7804.815,E2 7804.815} C_VEL
LIN {X 0,Y 160.682,Z 993.801,A -85,B 0,C 180,E1 7797.143,E2 7797.143} C_VEL
LIN {X 0,Y 168.58,Z 985.365,A -85,B 0,C 180,E1 7789.29,E2 7789.29} C_VEL
LIN {X 0,Y 177.61,Z 976.197,A -85,B 0,C 180,E1 7782.974,E2 7782.974} C_VEL
LIN {X 0,Y 188.558,Z 964.979,A -85,B 0,C 180,E1 7777.192,E2 7777.192} C_VEL
LIN {X 0,Y 200.591,Z 952.353,A -85,B 0,C 180,E1 7772.231,E2 7772.231} C_VEL
LIN {X 0,Y 213.017,Z 938.347,A -85,B 0,C 180,E1 7768.082,E2 7768.082} C_VEL
LIN {X 0,Y 226.194,Z 922.442,A -85,B 0,C 180,E1 7764.433,E2 7764.433} C_VEL
LIN {X 0,Y 238.188,Z 906.611,A -85,B 0,C 180,E1 7761.618,E2 7761.618} C_VEL
LIN {X 0,Y 250.692,Z 888.366,A -85,B 0,C 180,E1 7759.071,E2 7759.071} C_VEL
LIN {X 0,Y 262.379,Z 869.461,A -85,B 0,C 180,E1 7756.989,E2 7756.989} C_VEL
LIN {X 0,Y 273.044,Z 849.707,A -85,B 0,C 180,E1 7755.286,E2 7755.286} C_VEL
LIN {X 0,Y 283.139,Z 828.476,A -85,B 0,C 180,E1 7753.835,E2 7753.835} C_VEL
LIN {X 0,Y 291.585,Z 807.697,A -85,B 0,C 180,E1 7752.725,E2 7752.725} C_VEL
LIN {X 0,Y 299.456,Z 784.509,A -85,B 0,C 180,E1 7751.768,E2 7751.768} C_VEL
LIN {X 0,Y 305.878,Z 761.31,A -85,B 0,C 180,E1 7751.055,E2 7751.055} C_VEL
LIN {X 0,Y 310.644,Z 737.842,A -85,B 0,C 180,E1 7750.504,E2 7750.504} C_VEL
LIN {X 0,Y 314.793,Z 706.47,A -85,B 0,C 180,E1 7749.883,E2 7749.883} C_VEL
LIN {X 0,Y 327.118,Z 597.094,A -85,B 0,C 180,E1 7747.861,E2 7747.861} C_VEL
LIN {X 0,Y 322.678,Z 589.613,A -85,B 0,C 180,E1 7744.264,E2 7744.264} C_VEL
LIN {X 0,Y 319.536,Z 584.702,A -85,B 0,C 180,E1 7741.255,E2 7741.255} C_VEL
LIN {X 0,Y 317.04,Z 580.758,A -85,B 0,C 180,E1 7738.373,E2 7738.373} C_VEL
LIN {X 0,Y 314.222,Z 576.241,A -85,B 0,C 180,E1 7734.155,E2 7734.155} C_VEL
LIN {X 0,Y 311.777,Z 572.277,A -85,B 0,C 180,E1 7727.592,E2 7727.592} C_VEL
LIN {X 0,Y 311.551,Z 571.289,A -85,B 0,C 180,E1 7725.693,E2 7725.693} C_VEL
LIN {X 0,Y 311.668,Z 571.458,A -85,B 0,C 180,E1 7720.704,E2 7720.704} C_VEL
LIN {X 0,Y 313.74,Z 575.799,A -85,B 0,C 180,E1 7713.909,E2 7713.909} C_VEL
LIN {X 0,Y 314.653,Z 576.808,A -85,B 0,C 180,E1 7712.358,E2 7712.358} C_VEL
LIN {X 0,Y 317.92,Z 582.082,A -85,B 0,C 180,E1 7707.768,E2 7707.768} C_VEL
LIN {X 0,Y 320.924,Z 586.86,A -85,B 0,C 180,E1 7704.584,E2 7704.584} C_VEL
LIN {X 0,Y 324.666,Z 592.933,A -85,B 0,C 180,E1 7701.305,E2 7701.305} C_VEL
LIN {X 0,Y 326.753,Z 596.811,A -85,B 0,C 180,E1 7699.642,E2 7699.642} C_VEL
LIN {X 0,Y 312.337,Z 721.96,A -85,B 0,C 180,E1 7697.347,E2 7697.347} C_VEL
LIN {X 0,Y 307.955,Z 745.702,A -85,B 0,C 180,E1 7696.793,E2 7696.793} C_VEL
LIN {X 0,Y 302.47,Z 768.168,A -85,B 0,C 180,E1 7696.097,E2 7696.097} C_VEL
LIN {X 0,Y 295.75,Z 789.642,A -85,B 0,C 180,E1 7695.222,E2 7695.222} C_VEL
LIN {X 0,Y 287.451,Z 811.839,A -85,B 0,C 180,E1 7694.072,E2 7694.072} C_VEL
LIN {X 0,Y 278.829,Z 831.365,A -85,B 0,C 180,E1 7692.798,E2 7692.798} C_VEL
LIN {X 0,Y 267.926,Z 852.728,A -85,B 0,C 180,E1 7691.047,E2 7691.047} C_VEL
LIN {X 0,Y 256.879,Z 871.821,A -85,B 0,C 180,E1 7689.082,E2 7689.082} C_VEL
LIN {X 0,Y 245.09,Z 889.698,A -85,B 0,C 180,E1 7686.747,E2 7686.747} C_VEL
LIN {X 0,Y 232.501,Z 906.999,A -85,B 0,C 180,E1 7683.901,E2 7683.901} C_VEL
LIN {X 0,Y 220.592,Z 921.779,A -85,B 0,C 180,E1 7680.8,E2 7680.8} C_VEL
LIN {X 0,Y 207.178,Z 937.092,A -85,B 0,C 180,E1 7676.659,E2 7676.659} C_VEL
